// TwinCAT 3 PLC project main_program
// ProgramVersion: 3.1.4024.0
// libraries:
//   Tc2_MC2, * (Beckhoff Automation GmbH)
//   Tc2_Utilities, * (Beckhoff Automation GmbH)
//   Tc2_Standard, * (Beckhoff Automation GmbH)
//   Tc2_System, * (Beckhoff Automation GmbH)
//   Tc3_Module, * (Beckhoff Automation GmbH)
// project tree:
//   DUTs/ E_BiaxialState.TcDUT, E_PlcSystemStatus.TcDUT, E_SafetyState.TcDUT, E_SyncPoint.TcDUT, ST_settings.TcDUT (not stored), ST_MoveCommand.TcDUT, ST_SystemStatus.TcDUT
//   GVLs/ GVL_Axis.TcGVL (not stored), GVL_Persistent.TcGVL
//   / PlcTask.TcTTO (not stored)
//   POUs/ fb_MovementController.TcPOU, fb_AxisStatusPublisher.TcPOU, fb_BiaxialCoordinator.TcPOU, fb_safety.TcPOU, fb_StatusBuffer.TcPOU, MAIN.TcPOU
// real-time tasks:
//   TASK PlcTask: cycle T#10ms, priority 20, ADS port 350
// motion (NC):
//   TASK NC-Task 1 SAF: cycle T#2ms, priority 4, ADS port 501
//   TASK NC-Task 1 SVB: cycle T#10ms, priority 8, ADS port 511
//   AXIS xAxis (id 1)
//     Dynamic: Acceleration=150, Deceleration=150, Jerk=225
//     Velo: RefSearch=2, RefSync=5, SlowManual=5, FastManual=10, Maximum=100
//     OtherSettings: AllowMotionCmdToSlave=true
//     encoder EncType=19
//       EncPara: ScaleFactorNumerator=2, ScaleFactorDenominator=1048576, MaxCount=#xffffffff
//         SoftEndMaxControl: Range=10000
//         Inc: RefSearchInverse=true, RefPosition=-5
//     drive DrvType=16
//       DrvPara: MaxCount=#xffffffff, DriveControlDWord=#x00020100
//         Analog: TorqueSetpointScale=10, ScaleFactorActTorque=0.1
//         TimeComp: TaskDelayCycles=1
//     controller CtrType=1
//       CtrPara: PriorControlFactor=1
//         Observer: BandWidth=20
//   AXIS yAxis (id 2)
//     Dynamic: Acceleration=150, Deceleration=150, Jerk=225
//     Velo: RefSearch=2, RefSync=5, SlowManual=5, FastManual=10, Maximum=100
//     OtherSettings: AllowMotionCmdToSlave=true
//     encoder EncType=19
//       EncPara: ScaleFactorNumerator=2, ScaleFactorDenominator=1048576, MaxCount=#xffffffff
//         SoftEndMinControl: Enable=true
//         SoftEndMaxControl: Range=10000
//         Inc: RefSearchInverse=true, RefPosition=-5, RefMode=1
//     drive DrvType=16
//       DrvPara: MaxCount=#xffffffff, DriveControlDWord=#x00020100
//         Analog: TorqueSetpointScale=10, ScaleFactorActTorque=0.1
//         TimeComp: TaskDelayCycles=1
//     controller CtrType=1
//       CtrPara: PriorControlFactor=1
//         Observer: BandWidth=20
// I/O:
//   DEVICE Device 1 (EtherCAT), AmsNetId 5.85.113.174.2.1
//     Term 1 (EK1200) [EK1200-5000 EtherCAT Power supply (2A E-Bus)]
//       Term 2 (EL7062) [EL7062-0000 2Ch. Stepper motor output stage (48V, 3A)]
//       Term 3 (EL9510) [EL9510 Power supply terminal 10V]
//       Term 4 (EL3356-0020) [EL3356-0020 1Ch. Ana. Input Resistor Bridge Terminal, 24bit, High Precision, with calibration certificate]
//       Term 5 (EL3356-0020) [EL3356-0020 1Ch. Ana. Input Resistor Bridge Terminal, 24bit, High Precision, with calibration certificate]
//       Term 6 (EL9011) [EL9011 End Terminal]
// variable links:
//   NC-Task 1 SAF/Axes/xAxis <-> Device 1 (EtherCAT)/Term 1 (EK1200)/Term 2 (EL7062)
//     Drive/Inputs/In/nDataIn1 <-> DRV Following error actual value Channel 2/Following error actual value
//     Drive/Inputs/In/nDcOutputTime <-> InfoData/DcOutputShift
//     Drive/Inputs/In/nState1 <-> DRV Statusword Channel 2/Statusword
//     Drive/Inputs/In/nState2 <-> DRV Statusword Channel 2/Statusword @bit 8
//     Drive/Inputs/In/nState4 @bit 1 <-> WcState/InputToggle
//     Drive/Inputs/In/nState4 <-> WcState/WcState
//     Drive/Outputs/Out/nCtrl1 <-> DRV Controlword Channel 2/Controlword
//     Drive/Outputs/Out/nCtrl2 <-> DRV Controlword Channel 2/Controlword @bit 8
//     Drive/Outputs/Out/nDataOut1 <-> DRV Target position Channel 2/Target position
//     Enc/Inputs/In/nDataIn1 <-> FB Position Channel 2/Position
//     Enc/Inputs/In/nDcInputTime <-> InfoData/DcInputShift
//     Enc/Inputs/In/nState4 @bit 1 <-> WcState/InputToggle
//     Enc/Inputs/In/nState4 <-> WcState/WcState
//   NC-Task 1 SAF/Axes/yAxis <-> Device 1 (EtherCAT)/Term 1 (EK1200)/Term 2 (EL7062)
//     Drive/Inputs/In/nDataIn1 <-> DRV Following error actual value Channel 1/Following error actual value
//     Drive/Inputs/In/nDcOutputTime <-> InfoData/DcOutputShift
//     Drive/Inputs/In/nState1 <-> DRV Statusword Channel 1/Statusword
//     Drive/Inputs/In/nState2 <-> DRV Statusword Channel 1/Statusword @bit 8
//     Drive/Inputs/In/nState4 @bit 1 <-> WcState/InputToggle
//     Drive/Inputs/In/nState4 <-> WcState/WcState
//     Drive/Outputs/Out/nCtrl1 <-> DRV Controlword Channel 1/Controlword
//     Drive/Outputs/Out/nCtrl2 <-> DRV Controlword Channel 1/Controlword @bit 8
//     Drive/Outputs/Out/nDataOut1 <-> DRV Target position Channel 1/Target position
//     Enc/Inputs/In/nDataIn1 <-> FB Position Channel 1/Position
//     Enc/Inputs/In/nDcInputTime <-> InfoData/DcInputShift
//     Enc/Inputs/In/nState4 @bit 1 <-> WcState/InputToggle
//     Enc/Inputs/In/nState4 <-> WcState/WcState
//   main program/main program Instance <-> Device 1 (EtherCAT)/Term 1 (EK1200)/Term 2 (EL7062)
//     PlcTask Inputs/MAIN.nEndStopHx <-> DI Inputs Channel 2/Input 1
//     PlcTask Inputs/MAIN.nEndStopHy <-> DI Inputs Channel 1/Input 2
//     PlcTask Inputs/MAIN.nEndStopLx <-> DI Inputs Channel 1/Input 1
//     PlcTask Inputs/MAIN.nEndStopLy <-> DI Inputs Channel 2/Input 2
//   main program/main program Instance <-> Device 1 (EtherCAT)/Term 1 (EK1200)/Term 4 (EL3356-0020)
//     PlcTask Inputs/MAIN.nRawTenzoX <-> RMB Value (INT32)/Value
//   main program/main program Instance <-> Device 1 (EtherCAT)/Term 1 (EK1200)/Term 5 (EL3356-0020)
//     PlcTask Inputs/MAIN.nRawTenzoY <-> RMB Value (INT32)/Value
//   main program/main program Instance <-> NC-Task 1 SAF/Axes/xAxis
//     PlcTask Inputs/GVL_Axis.xAxis.NcToPlc <-> Outputs/ToPlc
//     PlcTask Outputs/GVL_Axis.xAxis.PlcToNc <-> Inputs/FromPlc
//   main program/main program Instance <-> NC-Task 1 SAF/Axes/yAxis
//     PlcTask Inputs/GVL_Axis.yAxis.NcToPlc <-> Outputs/ToPlc
//     PlcTask Outputs/GVL_Axis.yAxis.PlcToNc <-> Inputs/FromPlc

// ---- DUTs/E_BiaxialState.TcDUT
{attribute 'qualified_only'}
TYPE E_BiaxialState :
(
	Idle,
	Running,
	Aborting,
	Completing
);
END_TYPE

// ---- DUTs/E_PlcSystemStatus.TcDUT
{attribute 'qualified_only'}
TYPE E_PlcSystemStatus :
(
	Idle := 0,
	Error := 1,
	Homing := 2,
	Stopping := 3,
	Taring := 4,
	BasicMove := 5,
	ForceMode := 6,
	Pretension := 10,
	PreTestCyclic := 11,
	SingleTest := 20,
	CyclicTest := 21,
	PostTest := 30
);
END_TYPE

// ---- DUTs/E_SafetyState.TcDUT
TYPE E_SafetyState :
(
	Idle,
	RestoreReference,
	VerifyReference,
	Homing,
	MoveToZero,
	Complete,
	ProtectiveStop,
	ErrorStop
);
END_TYPE

// ---- DUTs/E_SyncPoint.TcDUT
{attribute 'qualified_only'}
TYPE E_SyncPoint :
(
	None := 0,
	PreTestDone := 1,
	LoadDone := 2,
	UnloadDone := 3,
	MainDone := 4,
	PostTestDone := 5,
	PretensionDone := 6
);
END_TYPE

// ---- DUTs/ST_MoveCommand.TcDUT
TYPE ST_MoveCommand :
	STRUCT
		// Mode 1: maintained jog
		fMoveVelocity : LREAL; // Signed jog velocity while bExecute is TRUE
		nJogLeaseCounter : UDINT; // Must change periodically while a jog is held

		// Mode 2: one PI-regulated force hold
		fTargetForce   : LREAL;
		fForceDuration : LREAL;
	
		// Command and service controls
		nMode       : INT;  // 1=jog, 2=force/time, 3=test sequence
		bExecute    : BOOL; // Start movement; maintained press signal for jog
		bHalt       : BOOL; // Panic stop
		bPower      : BOOL; // Maintained motor-enable request
		bReset      : BOOL; // Reset errors
		bHome       : BOOL; // Start homing sequence
		bStartTar   : BOOL; // Start tare sequence
		bSavePosition : BOOL; // Capture the current axis position while idle
		bRestorePosition : BOOL; // Return to the saved coordinate while idle
		fRestoreVelocity : LREAL; // Saved-position return speed [mm/s]

		// Optional force pre-conditioning sequence
		bIncludePreTest : BOOL;
		bPreTestOnly    : BOOL;  // Run pre-test and post-test without a main test
		nPreCycleCount  : INT;   // Number of force load/unload cycles, 0..50
		bPreloadEnabled : BOOL;  // Apply one force preload before the first cycle
		fPreloadValue   : LREAL; // Signed preload force [N]
		fPreCycleLoadValue : LREAL; // Signed repeated preconditioning load target [N]
		fPreUnloadValue : LREAL; // Signed force unload target [N]
		bPreUnloadToStart : BOOL; // Return to sequence-start position instead of force unload
		fPreTestRate     : LREAL; // Positive motor speed magnitude [mm/s]
		fPreTestForceTolerance : LREAL := 0.1; // [N], or negative for target-relative percent
		fPreloadHoldTime : LREAL := 0.0; // Hold time for the initial preload endpoint [s]
		fPreCycleHoldTime : LREAL := 0.0; // Hold time for cyclic pre-conditioning endpoints [s]

		// Main test settings
		fTestRate      : LREAL; // Positive motor speed magnitude [mm/s]
		fSingleForceTolerance : LREAL := 0.1; // [N], or negative for target-relative percent
		fSingleForceHoldTime : LREAL := 0.0; // Hold time for the single-test primary endpoint [s]
		fCyclicForceTolerance : LREAL := 0.1; // [N], or negative for target-relative percent
		fCyclicForceHoldTime : LREAL := 0.0; // Hold time for cyclic load/unload endpoints [s]

		// Test selection: >0=cyclic count, 0=single test
		nCycleCount : INT;
		nLoadMode   : INT;   // 1=displacement, 2=force
		fLoadValues : ARRAY[1..50] OF LREAL; // per-cycle level [mm] or signed force [N]
		nUnloadMode : INT;   // 1=displacement, 2=force
		fUnloadValues : ARRAY[1..50] OF LREAL; // per-cycle level [mm] or signed force [N]

		// Single test (nMode=3, nCycleCount=0); criterion 2 is optional OR
		nStop1Mode         : INT;   // 0=off, 1=displacement, 2=force
		fStop1Value        : LREAL;
		nStop2Mode         : INT;   // 0=off, 1=displacement, 2=force, 3=rupture
		fStop2Value        : LREAL;

		// 0=stay, 1=saved position, 2=sequence start,
		// 3=pre-test final position, 4=unload to zero force
		nPostTestMode : INT;
	END_STRUCT
END_TYPE

// ---- DUTs/ST_SystemStatus.TcDUT
TYPE ST_SystemStatus :
	STRUCT
		fPosBuffer   : ARRAY[1..50] OF LREAL; // Circular display-position samples
		fTenzoBuffer : ARRAY[1..50] OF LREAL; // Circular force samples
		nBufferHead  : INT := 50;             // Index of latest completely written sample
		nSampleCounter    : UDINT := 0;       // Wrapping sample counter for drop detection
		nOperationCounter : UDINT := 0;       // Incremented after each completed motion command
		nInterfaceVersion : UDINT := 7;       // MATLAB/PLC ADS contract version
		fTenzoTarOffset   : LREAL := 0.0;     // Calculated tar offset
		fActPosition : LREAL := 0.0;          // Display position (50 mm - NC position)
		
		bWorking     : BOOL;                   // PLC occupied; do not send a new test
		bTarWorking  : BOOL;                   // PLC is calculating tare
		bError       : BOOL;                   // Latched application or motion error
		nErrorCode   : UDINT := 0;             // Application error code (0 = no error)
		nAxisErrorID : UDINT := 0;             // Native TwinCAT/NC error ID
		bPowered     : BOOL;                   // Axis power is enabled
		bHoming      : BOOL;                   // Homing command is active
		bHomed       : BOOL;                   // NC axis reports a valid home reference
		bStopped     : BOOL;                   // Axis is at standstill
		bSavedPositionValid : BOOL;            // A return-to-saved reference is available
		nSystemStatus : INT := 0;              // High-level numeric system status
	END_STRUCT
END_TYPE

// ---- GVLs/GVL_Persistent.TcGVL
{attribute 'qualified_only'}
VAR_GLOBAL PERSISTENT
	// Last valid incremental-axis coordinates
	fLastPositionX      : LREAL;
	fLastPositionY      : LREAL;
	bLastPositionValidX : BOOL;
	bLastPositionValidY : BOOL;
END_VAR

// ---- POUs/fb_MovementController.TcPOU
FUNCTION_BLOCK fb_MovementController
VAR_INPUT
	fForce        : LREAL; // Actual force
	fActPosition  : LREAL; // Absolute NC position
	bPowerState   : BOOL;  // Actual power on state
	bHaltDone     : BOOL;  // Motor stopped
	bAxisStopped  : BOOL;  // Fresh safety/NC standstill state
	bSafetyError  : BOOL;
	bProtectiveStop : BOOL;
	bExternalBusy : BOOL;
	bReferenceValid : BOOL; // Current home/reference belongs to this coordinate system
	bInvalidateSavedPosition : BOOL; // Home request invalidates saved absolute coordinates
	bSyncEnabled  : BOOL;  // TRUE only for a PLC-owned biaxial test
	bSyncRelease  : BOOL;  // Shared barrier release from MAIN
	bSyncAbort    : BOOL;  // Stop this axis when the synchronized peer aborts
	bSyncSingleComplete : BOOL; // Peer reached its biaxial Single endpoint
	stSettings    : ST_Settings;
END_VAR

VAR_OUTPUT
	fTestStartPos : LREAL := 0.0; // position where test started
	stateHalt   : BOOL; // Request a controlled stop
	bBusy       : BOOL; // System is processing a test or stopping
	bError      : BOOL; // Latched application/motion error
	nErrorCode  : UDINT;
	nAxisErrorID: UDINT;
	nOperationCounter : UDINT;
	bSavedPositionValid : BOOL;
	nSystemStatus : INT; // High-level numeric system status exposed through ADS
	nSyncPoint : BYTE; // E_SyncPoint: 0 none through 6 pretension
	nSyncCycle : INT;  // Cycle associated with the current sync point
	bPeerAbortRequest : BOOL; // Abort synchronized peer while local relief continues
END_VAR

VAR
	// Movement FBs
	fbMC_MoveRelative1 : MC_MoveRelative;
	fbMC_MoveVelocity  : MC_MoveVelocity;
	
	// Shared help vars
	nSeqState    : INT; // Current sequence state
	
	// mode 1
	fTargetDist1 : LREAL;
	fTargetVel1  : LREAL;
	
	// mode 2/3 vel movement
	bExecuteVelMove : BOOL;
    fCmdVelocity    : LREAL;
    mcDirection     : MC_Direction;
	
	// mode 2/3 help vars
	fTargetForce          : LREAL; // Wanted F
    fForceError           : LREAL; // Regulation error
    fForceErrorIntegral   : LREAL; // Integ of error
	fMode2HoldElapsed     : LREAL; // Accumulated time inside force tolerance
	fLastSentVelocity   : LREAL;    // Tracks last updated velocity to prevent NC spamming
	fPendingVelocity   : LREAL;
	mcPendingDirection : MC_Direction;
	nVelocityState     : INT;
	nVelocityUpdateCounter : INT;
	fForceRegMaxVelocity : LREAL; // Mode-3 P regulator speed limit
	fForceRegMinVelocity : LREAL; // Mode-3 low-speed hold deadband
	bResetRequested : BOOL;
	bOperationCompleted : BOOL;

	// Saved/reference positions
	fSavedPosition      : LREAL;
	fPreTestFinalPos    : LREAL;
	rtSavePosition      : R_TRIG;
	rtRestorePosition   : R_TRIG;
	rtSyncAbort         : R_TRIG;
	fbJogLease          : TON;
	nLastJogLeaseCounter : UDINT;
	bJogLeaseRenewed    : BOOL;

	// Generic endpoint engine for test-sequence mode 3
	nCurrentCycle           : INT;
	nCurrentPreCycle        : INT;
	nAfterEndpointState     : INT;
	fEndpointTargetPosition : LREAL;
	fEndpointTargetForce    : LREAL;
	fEndpointRate           : LREAL;
	fEndpointTolerance      : LREAL;
	fEndpointHoldTime       : LREAL;
	fEndpointStartError     : LREAL;
	fEndpointCurrentError   : LREAL;
	fForceHoldElapsed       : LREAL;
	fPositionHoldElapsed    : LREAL;
	nLoadDirection          : INT;
	nLastMotionDirection    : INT;
	nReliefSourceDirection  : INT;
	nEndpointSyncPoint      : BYTE;
	nEndpointSyncCycle      : INT;
	bForceEndpointReady     : BOOL;
	bZeroForceUnload        : BOOL; // Post-test unload must not reverse across zero

	// Optional OR criterion for the single test
	bSinglePrimaryActive  : BOOL;
	bSingleStopReached    : BOOL;
	fStop2TargetPosition  : LREAL;
	fStop2StartError      : LREAL;
	fStop2CurrentError    : LREAL;
	fSingleStartForce     : LREAL;
	fSinglePeakForce      : LREAL;
	bSingleRuptureArmed   : BOOL;
	
END_VAR

VAR CONSTANT
	// Task and controller constants
	CYCLE_TIME : LREAL := 0.01; // dt of plc
	VELOCITY_UPDATE_DELTA : LREAL := 0.1;
	VELOCITY_UPDATE_CYCLES : INT := 10;
	FORCE_REG_MIN_SPEED_FRACTION : LREAL := 0.01;
	POSITION_EPSILON : LREAL := 0.000001;
	FORCE_POLARITY : INT := -1;
	STATUS_IDLE : INT := 0;
	STATUS_STOPPING : INT := 3;
	STATUS_BASIC_MOVE : INT := 5;
	STATUS_FORCE_MODE : INT := 6;
	STATUS_PRETENSION : INT := 10;
	STATUS_PRETEST_CYCLIC : INT := 11;
	STATUS_SINGLE_TEST : INT := 20;
	STATUS_CYCLIC_TEST : INT := 21;
	STATUS_POSTTEST : INT := 30;
	SYNC_NONE : BYTE := 0;
	SYNC_PRETEST_DONE : BYTE := 1;
	SYNC_LOAD_DONE : BYTE := 2;
	SYNC_UNLOAD_DONE : BYTE := 3;
	SYNC_MAIN_DONE : BYTE := 4;
	SYNC_POSTTEST_DONE : BYTE := 5;
	SYNC_PRETENSION_DONE : BYTE := 6;
	STATE_IDLE : INT := 0;
	STATE_MODE_START : INT := 1;
	STATE_MODE_RUN : INT := 2;
	STATE_PRELOAD : INT := 10;
	STATE_CAPTURE_TEST_START : INT := 11;
	STATE_PRE_CYCLE_LOAD : INT := 12;
	STATE_PRE_CYCLE_UNLOAD : INT := 13;
	STATE_PRE_CYCLE_NEXT : INT := 14;
	STATE_CAPTURE_PRETEST_FINAL : INT := 18;
	STATE_PRETEST_BARRIER : INT := 19;
	STATE_SELECT_MAIN_TEST : INT := 20;
	STATE_SECONDARY_BARRIER : INT := 49;
	STATE_POSTTEST_SELECT : INT := 50;
	STATE_POSTTEST_WAIT_STOP : INT := 51;
	STATE_POSTTEST_BARRIER : INT := 54;
	STATE_OPERATION_COMPLETE : INT := 55;
	STATE_RESTORE_COMPLETE : INT := 56;
	STATE_CYCLIC_LOAD : INT := 100;
	STATE_CYCLIC_UNLOAD : INT := 110;
	STATE_CYCLIC_NEXT : INT := 120;
	STATE_CYCLIC_COMPLETE : INT := 121;
	STATE_SINGLE_START : INT := 200;
	STATE_SINGLE_WAIT_STOP : INT := 220;
	STATE_POSITION_PREPARE : INT := 300;
	STATE_POSITION_EXECUTE : INT := 301;
	STATE_POSITION_WAIT : INT := 302;
	STATE_POSITION_HOLD : INT := 303;
	STATE_POSITION_BARRIER : INT := 304;
	STATE_FORCE_PREPARE : INT := 310;
	STATE_FORCE_EXECUTE : INT := 311;
	STATE_FORCE_WAIT_TOLERANCE : INT := 312;
	STATE_FORCE_WAIT_STOP : INT := 313;
	STATE_FORCE_HOLD : INT := 314;
	STATE_FORCE_EXIT_WAIT_STOP : INT := 315;
	STATE_FORCE_READY_WAIT_STOP : INT := 316;
	STATE_ABORT_STOPPING : INT := 900;
	STATE_RELIEF_WAIT_STOP : INT := 910;
	STATE_RELIEF_START : INT := 911;
	STATE_RELIEF_WAIT_MOVE : INT := 912;
	STATE_ERROR_STOPPING : INT := 998;
	STATE_ERROR_LATCHED : INT := 999;
	ERROR_UNSUPPORTED_MODE : UDINT := 2001;
	ERROR_SAVED_POSITION_UNAVAILABLE : UDINT := 2002;
	ERROR_UNSUPPORTED_ENDPOINT : UDINT := 2003;
	ERROR_UNSUPPORTED_POST_ACTION : UDINT := 2005;
	ERROR_POWER_UNAVAILABLE : UDINT := 2006;
	ERROR_INVALID_CONFIGURATION : UDINT := 2007;
	ERROR_COMMAND_CONFLICT : UDINT := 2008;
	ERROR_INVALID_RUNTIME_VALUE : UDINT := 2009;
	ERROR_JOG_LEASE_EXPIRED : UDINT := 2011;
	ERROR_VELOCITY_LIMIT : UDINT := 2012;
	ERROR_RELIEF_COMPLETED : UDINT := 2101;
	ERROR_RELIEF_DIRECTION_UNKNOWN : UDINT := 2102;
	ERROR_RELATIVE_MOVE : UDINT := 2201;
	ERROR_VELOCITY_MOVE : UDINT := 2203;
END_VAR

VAR_IN_OUT
	Axis          : AXIS_REF;
	stMoveCommand : ST_MoveCommand;
END_VAR


// =========================================================
//                    Saved position
// =========================================================

rtSavePosition(CLK := stMoveCommand.bSavePosition);
rtRestorePosition(CLK := stMoveCommand.bRestorePosition);
rtSyncAbort(CLK := bSyncEnabled AND bSyncAbort);

// Saved positions are absolute NC coordinates. A new home/reference changes
// their meaning, so discard them as soon as homing starts or reference is lost.
IF bInvalidateSavedPosition OR NOT bReferenceValid THEN
	bSavedPositionValid := FALSE;
END_IF

IF rtSavePosition.Q AND nSeqState = STATE_IDLE AND NOT bExternalBusy AND
	bReferenceValid AND bAxisStopped THEN
	fSavedPosition := fActPosition;
	bSavedPositionValid := TRUE;
END_IF

// A maintained jog must be renewed by the ADS owner. The monotonically
// increasing counter makes a stale TRUE bExecute harmless after owner loss.
bJogLeaseRenewed := nSeqState = STATE_MODE_RUN AND
	stMoveCommand.nMode = 1 AND
	stMoveCommand.nJogLeaseCounter <> nLastJogLeaseCounter;
IF bJogLeaseRenewed THEN
	nLastJogLeaseCounter := stMoveCommand.nJogLeaseCounter;
END_IF
fbJogLease(
	IN := nSeqState = STATE_MODE_RUN AND stMoveCommand.nMode = 1 AND
		NOT bJogLeaseRenewed,
	PT := T#750MS);
IF fbJogLease.Q AND NOT bError AND NOT bSafetyError THEN
	stMoveCommand.bExecute := FALSE;
	SetError(
		nCode := ERROR_JOG_LEASE_EXPIRED,
		nNativeErrorID := 0,
		bRequestHalt := TRUE);
END_IF

// =========================================================
//                      Error handling
// =========================================================

IF stMoveCommand.bReset THEN
	bResetRequested := TRUE;
END_IF

IF bResetRequested AND bError AND NOT bSafetyError THEN
	bError := FALSE;
	nErrorCode := 0;
	nAxisErrorID := 0;
	nSeqState := STATE_IDLE;
	stateHalt := FALSE;
	bResetRequested := FALSE;
ELSIF bResetRequested AND NOT bError AND NOT bSafetyError THEN
	IF nSeqState = STATE_ERROR_LATCHED THEN
		nSeqState := STATE_IDLE;
	END_IF
	bResetRequested := FALSE;
END_IF

// Operator and safety stops abort the sequence without running post-test.
IF stMoveCommand.bHalt OR (bProtectiveStop AND NOT stateHalt) OR
	rtSyncAbort.Q THEN
	IF stMoveCommand.bHalt THEN
		stMoveCommand.bHalt := FALSE;
	END_IF
	stMoveCommand.bExecute := FALSE;
	ClearActiveCommand();
	stateHalt := TRUE;
	nSeqState := STATE_ABORT_STOPPING;
END_IF

// A safety-owned error cancels local motion without issuing another halt.
IF bSafetyError THEN
	stMoveCommand.bExecute := FALSE;
	ClearActiveCommand();
	stateHalt := FALSE;
	nSeqState := STATE_ERROR_LATCHED;
END_IF

// Latch motion-function-block and sensor errors.
IF NOT bError AND NOT bSafetyError THEN
	IF fbMC_MoveRelative1.Error THEN
		bError := TRUE;
		nErrorCode := ERROR_RELATIVE_MOVE;
		nAxisErrorID := fbMC_MoveRelative1.ErrorID;
	ELSIF fbMC_MoveVelocity.Error THEN
		bError := TRUE;
		nErrorCode := ERROR_VELOCITY_MOVE;
		nAxisErrorID := fbMC_MoveVelocity.ErrorID;
	ELSIF nSeqState > STATE_IDLE AND
		nSeqState < STATE_ABORT_STOPPING AND
		NOT ((fForce = fForce) AND ABS(fForce) < 1.0E300) THEN
		bError := TRUE;
		nErrorCode := ERROR_INVALID_RUNTIME_VALUE;
	END_IF
END_IF

// Runtime overforce response: halt, make one fixed relative release move, then abort.
IF NOT bError AND NOT bSafetyError AND
	nSeqState > STATE_IDLE AND nSeqState < STATE_ABORT_STOPPING AND
	ABS(fForce) >= stSettings.fMaxForce THEN
	IF Axis.Status.PositiveDirection THEN
		nReliefSourceDirection := 1;
	ELSIF Axis.Status.NegativeDirection THEN
		nReliefSourceDirection := -1;
	ELSIF stMoveCommand.nMode = 3 AND nLoadDirection <> 0 THEN
		nReliefSourceDirection := nLoadDirection;
	ELSE
		nReliefSourceDirection := nLastMotionDirection;
	END_IF
	fbMC_MoveRelative1.Execute := FALSE;
	bExecuteVelMove := FALSE;
	bSinglePrimaryActive := FALSE;
	bForceEndpointReady := FALSE;
	nSyncPoint := SYNC_NONE;
	nSyncCycle := 0;
	stateHalt := TRUE;
	nSeqState := STATE_RELIEF_WAIT_STOP;
END_IF

IF bError AND nSeqState <> STATE_ERROR_STOPPING AND
	nSeqState <> STATE_ERROR_LATCHED THEN
	stMoveCommand.bExecute := FALSE;
	ClearActiveCommand();
	stateHalt := TRUE;
	nSeqState := STATE_ERROR_STOPPING;
END_IF

IF bError THEN
	stMoveCommand.bExecute := FALSE;
END_IF

IF stMoveCommand.bExecute AND bExternalBusy THEN
	stMoveCommand.bExecute := FALSE;
	bError := TRUE;
	nErrorCode := ERROR_COMMAND_CONFLICT;
END_IF

IF stMoveCommand.bExecute AND NOT bPowerState THEN
	stMoveCommand.bExecute := FALSE;
	bError := TRUE;
	nErrorCode := ERROR_POWER_UNAVAILABLE;
END_IF

// Finish operator/error stops.
IF (nSeqState = STATE_ABORT_STOPPING OR
	nSeqState = STATE_ERROR_STOPPING) AND bHaltDone THEN
	stateHalt := FALSE;
	IF nSeqState = STATE_ERROR_STOPPING THEN
		nSeqState := STATE_ERROR_LATCHED;
	ELSE
		nSeqState := STATE_IDLE;
	END_IF
END_IF

// Overforce release sequence. FB1 is reused with aborting buffer mode.
CASE nSeqState OF
	STATE_RELIEF_WAIT_STOP:
		IF bHaltDone THEN
			stateHalt := FALSE;
			IF nReliefSourceDirection = 0 THEN
				bError := TRUE;
				nErrorCode := ERROR_RELIEF_DIRECTION_UNKNOWN;
				nSeqState := STATE_ERROR_LATCHED;
			ELSE
				fTargetDist1 := -INT_TO_LREAL(nReliefSourceDirection) *
					ABS(stSettings.fForceReliefDistance);
				fTargetVel1 := ABS(stSettings.fForceReliefVelocity);
				fbMC_MoveRelative1.Execute := FALSE;
				nSeqState := STATE_RELIEF_START;
			END_IF
		END_IF

	STATE_RELIEF_START:
		fbMC_MoveRelative1.Execute := TRUE;
		nSeqState := STATE_RELIEF_WAIT_MOVE;

	STATE_RELIEF_WAIT_MOVE:
		IF fbMC_MoveRelative1.Done THEN
			fbMC_MoveRelative1.Execute := FALSE;
			bError := TRUE;
			nErrorCode := ERROR_RELIEF_COMPLETED;
			nAxisErrorID := 0;
			nSeqState := STATE_ERROR_LATCHED;
		END_IF
END_CASE

// Saved-position restore is a service operation and is independent of nMode.
IF rtRestorePosition.Q AND nSeqState = STATE_IDLE AND
	NOT bError AND NOT bSafetyError THEN
	IF bExternalBusy THEN
		stMoveCommand.bExecute := FALSE;
		SetError(
			nCode := ERROR_COMMAND_CONFLICT,
			nNativeErrorID := 0,
			bRequestHalt := TRUE);
	ELSIF NOT bPowerState THEN
		stMoveCommand.bExecute := FALSE;
		SetError(
			nCode := ERROR_POWER_UNAVAILABLE,
			nNativeErrorID := 0,
			bRequestHalt := TRUE);
	ELSIF NOT bReferenceValid OR NOT bSavedPositionValid THEN
		stMoveCommand.bExecute := FALSE;
		SetError(
			nCode := ERROR_SAVED_POSITION_UNAVAILABLE,
			nNativeErrorID := 0,
			bRequestHalt := TRUE);
	ELSIF NOT ((stMoveCommand.fRestoreVelocity =
		stMoveCommand.fRestoreVelocity) AND
		ABS(stMoveCommand.fRestoreVelocity) > 0.0 AND
		ABS(stMoveCommand.fRestoreVelocity) < 1.0E300) THEN
		stMoveCommand.bExecute := FALSE;
		SetError(
			nCode := ERROR_INVALID_RUNTIME_VALUE,
			nNativeErrorID := 0,
			bRequestHalt := TRUE);
	ELSIF ABS(stMoveCommand.fRestoreVelocity) > ABS(stSettings.fMaxVelocity) THEN
		stMoveCommand.bExecute := FALSE;
		SetError(
			nCode := ERROR_VELOCITY_LIMIT,
			nNativeErrorID := 0,
			bRequestHalt := TRUE);
	ELSE
		fTestStartPos := fActPosition;
		nSystemStatus := STATUS_BASIC_MOVE;
		nLoadDirection := 0;
		nLastMotionDirection := 0;
		nReliefSourceDirection := 0;
		PreparePositionEndpoint(
			fTargetPosition := fSavedPosition,
			fRate := stMoveCommand.fRestoreVelocity,
			fHoldTime := 0.0,
			nTargetSyncPoint := SYNC_NONE,
			nTargetSyncCycle := 0,
			nNextState := STATE_RESTORE_COMPLETE);
	END_IF
END_IF

// =========================================================
//                      Mode switcher
// =========================================================

// In a biaxial Single test, either axis endpoint completes both axes.
IF bSinglePrimaryActive AND bSyncSingleComplete THEN
	fbMC_MoveRelative1.Execute := FALSE;
	bExecuteVelMove := FALSE;
	bSinglePrimaryActive := FALSE;
	stateHalt := TRUE;
	nSeqState := STATE_SINGLE_WAIT_STOP;
END_IF

IF NOT bError AND NOT bSafetyError AND
	nSeqState < STATE_ABORT_STOPPING THEN
	IF nSeqState >= STATE_POSITION_PREPARE AND
		nSeqState <= STATE_POSITION_BARRIER THEN
		positionEndpoint();
	ELSIF nSeqState >= STATE_FORCE_PREPARE AND
		nSeqState <= STATE_FORCE_READY_WAIT_STOP THEN
		forceEndpoint();
	ELSIF nSeqState = STATE_RESTORE_COMPLETE THEN
		testSequence();
	ELSE
		CASE stMoveCommand.nMode OF
			1: mode1();
			2: mode2();
			3: testSequence();
		ELSE
			IF stMoveCommand.bExecute THEN
				stMoveCommand.bExecute := FALSE;
				bError := TRUE;
				nErrorCode := ERROR_UNSUPPORTED_MODE;
			END_IF
		END_CASE
	END_IF
END_IF

// =========================================================
//                      Motion calls
// =========================================================

fbMC_MoveRelative1(
	Axis := Axis,
	Distance := fTargetDist1,
	Velocity := MIN(ABS(fTargetVel1), ABS(stSettings.fMaxVelocity)),
	BufferMode := MC_Aborting);

fbMC_MoveVelocity(
	Axis := Axis,
	Execute := bExecuteVelMove,
	Velocity := MIN(ABS(fCmdVelocity), ABS(stSettings.fMaxVelocity)),
	Direction := mcDirection,
	BufferMode := MC_Aborting);

IF Axis.Status.PositiveDirection THEN
	nLastMotionDirection := 1;
ELSIF Axis.Status.NegativeDirection THEN
	nLastMotionDirection := -1;
END_IF

// =========================================================
//                         Outputs
// =========================================================

IF nSeqState = STATE_IDLE THEN
	nSystemStatus := STATUS_IDLE;
ELSIF nSeqState >= STATE_ABORT_STOPPING THEN
	nSystemStatus := STATUS_STOPPING;
END_IF

// Expose a newly entered relief state in this scan
bPeerAbortRequest := nSeqState >= STATE_RELIEF_WAIT_STOP AND
	nSeqState <= STATE_RELIEF_WAIT_MOVE;

bBusy := nSeqState > STATE_IDLE AND
	nSeqState <> STATE_ERROR_LATCHED;

IF bOperationCompleted THEN
	nOperationCounter := nOperationCounter + 1;
	bOperationCompleted := FALSE;
END_IF

METHOD ClearActiveCommand

fbMC_MoveRelative1.Execute := FALSE;
bExecuteVelMove := FALSE;
bSinglePrimaryActive := FALSE;
bForceEndpointReady := FALSE;
bZeroForceUnload := FALSE;
fPositionHoldElapsed := 0.0;
nSyncPoint := SYNC_NONE;
nSyncCycle := 0;
END_METHOD

ACTION forceEndpoint:

CASE nSeqState OF
	STATE_FORCE_PREPARE:
		bExecuteVelMove := FALSE;
		fForceHoldElapsed := 0.0;
		bForceEndpointReady := FALSE;
		nSyncPoint := SYNC_NONE;
		nSyncCycle := 0;
		fEndpointStartError := fEndpointTargetForce - fForce;
		nVelocityState := 0;
		nVelocityUpdateCounter := VELOCITY_UPDATE_CYCLES;
		fLastSentVelocity := 0.0;
		fForceRegMaxVelocity := MIN(
			ABS(fEndpointRate),
			ABS(stSettings.fMaxVelocity));
		// Keep the anti-chatter floor small enough that force endpoints settle
		// near the requested goal instead of at the edge of a 10% speed band.
		fForceRegMinVelocity := fForceRegMaxVelocity *
			FORCE_REG_MIN_SPEED_FRACTION;
		fCmdVelocity := ABS(fEndpointRate);
		IF fEndpointStartError * INT_TO_LREAL(FORCE_POLARITY) >= 0.0 THEN
			mcDirection := MC_Positive_Direction;
			nLoadDirection := 1;
			nLastMotionDirection := 1;
		ELSE
			mcDirection := MC_Negative_Direction;
			nLoadDirection := -1;
			nLastMotionDirection := -1;
		END_IF
		IF ABS(fEndpointStartError) <= fEndpointTolerance THEN
			stateHalt := TRUE;
			nVelocityState := 3;
			nSeqState := STATE_FORCE_WAIT_STOP;
		ELSE
			nSeqState := STATE_FORCE_EXECUTE;
		END_IF

	STATE_FORCE_EXECUTE: // Trigger constant-speed force approach.
		bExecuteVelMove := TRUE;
		nVelocityState := 1;
		nSeqState := STATE_FORCE_WAIT_TOLERANCE;

	STATE_FORCE_WAIT_TOLERANCE:
		fEndpointCurrentError := fEndpointTargetForce - fForce;
		IF ABS(fEndpointCurrentError) <= fEndpointTolerance OR
			(fEndpointStartError > 0.0 AND fEndpointCurrentError <= 0.0) OR
			(fEndpointStartError < 0.0 AND fEndpointCurrentError >= 0.0) THEN
			bExecuteVelMove := FALSE;
			stateHalt := TRUE;
			nVelocityState := 3;
			nSeqState := STATE_FORCE_WAIT_STOP;
		END_IF

	STATE_FORCE_WAIT_STOP:
		IF bHaltDone THEN
			stateHalt := FALSE;
			nVelocityState := 4;
			IF bZeroForceUnload THEN
				IF bSyncEnabled AND nEndpointSyncPoint <> SYNC_NONE THEN
					bForceEndpointReady := TRUE;
					nSyncPoint := nEndpointSyncPoint;
					nSyncCycle := nEndpointSyncCycle;
					nSeqState := STATE_FORCE_HOLD;
				ELSE
					bZeroForceUnload := FALSE;
					nSeqState := nAfterEndpointState;
				END_IF
			ELSE
				nVelocityUpdateCounter := VELOCITY_UPDATE_CYCLES;
				fLastSentVelocity := 0.0;
				nSeqState := STATE_FORCE_HOLD;
			END_IF
		END_IF

	STATE_FORCE_HOLD: // P-regulate while the timer runs and the peer catches up.
		IF bZeroForceUnload AND NOT bSyncRelease THEN
			// Wait at standstill for the other axis; never reload across zero.
			bExecuteVelMove := FALSE;
		ELSIF bForceEndpointReady AND bSyncRelease THEN
			bExecuteVelMove := FALSE;
			bForceEndpointReady := FALSE;
			bZeroForceUnload := FALSE;
			nSyncPoint := SYNC_NONE;
			nSyncCycle := 0;
			nEndpointSyncPoint := SYNC_NONE;
			IF nVelocityState = 4 THEN
				nSeqState := nAfterEndpointState;
			ELSE
				stateHalt := TRUE;
				nVelocityState := 3;
				nSeqState := STATE_FORCE_EXIT_WAIT_STOP;
			END_IF
		ELSE
			fForceError := fEndpointTargetForce - fForce;

			// Proportional correction begins only after the initial
			// constant-speed approach has reached the endpoint.
			fCmdVelocity := (fForceError * stSettings.fKp) *
				INT_TO_LREAL(FORCE_POLARITY);
			fCmdVelocity := LIMIT(
				-fForceRegMaxVelocity,
				fCmdVelocity,
				fForceRegMaxVelocity);
			fPendingVelocity := ABS(fCmdVelocity);
			IF fCmdVelocity >= 0.0 THEN
				mcPendingDirection := MC_Positive_Direction;
			ELSE
				mcPendingDirection := MC_Negative_Direction;
			END_IF
			IF nVelocityUpdateCounter < VELOCITY_UPDATE_CYCLES THEN
				nVelocityUpdateCounter := nVelocityUpdateCounter + 1;
			END_IF

			// Tiny corrections are replaced by a powered position hold.
			IF fPendingVelocity <= fForceRegMinVelocity THEN
				bExecuteVelMove := FALSE;
				IF nVelocityState <> 3 AND nVelocityState <> 4 THEN
					stateHalt := TRUE;
					nVelocityState := 3;
				ELSIF nVelocityState = 3 AND bHaltDone THEN
					stateHalt := FALSE;
					nVelocityState := 4;
				END_IF
			ELSIF nVelocityState = 3 THEN
				IF bHaltDone THEN
					stateHalt := FALSE;
					nVelocityState := 0;
				END_IF
			ELSIF nVelocityState = 4 THEN
				nVelocityState := 0;
			ELSIF nVelocityState = 2 THEN
				fCmdVelocity := fPendingVelocity;
				mcDirection := mcPendingDirection;
				IF mcDirection = MC_Positive_Direction THEN
					nLoadDirection := 1;
					nLastMotionDirection := 1;
				ELSE
					nLoadDirection := -1;
					nLastMotionDirection := -1;
				END_IF
				bExecuteVelMove := TRUE;
				fLastSentVelocity := fCmdVelocity;
				nVelocityUpdateCounter := 0;
				nVelocityState := 1;
			ELSE
				IF nVelocityState = 0 THEN
					fCmdVelocity := fPendingVelocity;
					mcDirection := mcPendingDirection;
					IF mcDirection = MC_Positive_Direction THEN
						nLoadDirection := 1;
						nLastMotionDirection := 1;
					ELSE
						nLoadDirection := -1;
						nLastMotionDirection := -1;
					END_IF
					bExecuteVelMove := TRUE;
					fLastSentVelocity := fCmdVelocity;
					nVelocityUpdateCounter := 0;
					nVelocityState := 1;
				ELSIF nVelocityUpdateCounter >=
					VELOCITY_UPDATE_CYCLES AND
					(ABS(fPendingVelocity - fLastSentVelocity) >=
						fForceRegMinVelocity OR
					 mcPendingDirection <> mcDirection) THEN
					bExecuteVelMove := FALSE;
					nVelocityState := 2;
				END_IF
			END_IF

			// Hold time is accumulated only inside tolerance. Excursions
			// pause it and withdraw readiness without resetting elapsed time.
			IF ABS(fForceError) <= fEndpointTolerance THEN
				IF NOT bForceEndpointReady THEN
					fForceHoldElapsed := fForceHoldElapsed + CYCLE_TIME;
					IF fForceHoldElapsed >= fEndpointHoldTime THEN
						IF bSyncEnabled AND
							nEndpointSyncPoint <> SYNC_NONE THEN
							// Publish barrier readiness only at confirmed
							// standstill. Otherwise both axes could be released
							// while one is still executing a correction.
							bExecuteVelMove := FALSE;
							IF nVelocityState = 4 THEN
								bForceEndpointReady := TRUE;
								nSyncPoint := nEndpointSyncPoint;
								nSyncCycle := nEndpointSyncCycle;
							ELSE
								stateHalt := TRUE;
								nVelocityState := 3;
								nSeqState :=
									STATE_FORCE_READY_WAIT_STOP;
							END_IF
						ELSE
							bExecuteVelMove := FALSE;
							IF nVelocityState = 4 THEN
								nSeqState := nAfterEndpointState;
							ELSE
								stateHalt := TRUE;
								nVelocityState := 3;
								nSeqState :=
									STATE_FORCE_EXIT_WAIT_STOP;
							END_IF
						END_IF
					END_IF
				END_IF
			ELSIF bForceEndpointReady THEN
				bForceEndpointReady := FALSE;
				nSyncPoint := SYNC_NONE;
				nSyncCycle := 0;
			END_IF
		END_IF

	STATE_FORCE_EXIT_WAIT_STOP:
		bExecuteVelMove := FALSE;
		IF bHaltDone THEN
			stateHalt := FALSE;
			nVelocityState := 4;
			nSeqState := nAfterEndpointState;
		END_IF

	STATE_FORCE_READY_WAIT_STOP:
		bExecuteVelMove := FALSE;
		IF bHaltDone THEN
			stateHalt := FALSE;
			nVelocityState := 4;
			fForceError := fEndpointTargetForce - fForce;
			IF ABS(fForceError) <= fEndpointTolerance THEN
				bForceEndpointReady := TRUE;
				nSyncPoint := nEndpointSyncPoint;
				nSyncCycle := nEndpointSyncCycle;
			END_IF
			nSeqState := STATE_FORCE_HOLD;
		END_IF
END_CASE
END_ACTION

ACTION mode1:

// =========================================================
//                  Mode 1: Maintained jog
// =========================================================

CASE nSeqState OF
	STATE_IDLE:
		IF stMoveCommand.bExecute THEN
			IF NOT ((stMoveCommand.fMoveVelocity =
				stMoveCommand.fMoveVelocity) AND
				ABS(stMoveCommand.fMoveVelocity) > 0.0 AND
				ABS(stMoveCommand.fMoveVelocity) < 1.0E300) THEN
				stMoveCommand.bExecute := FALSE;
				SetError(
					nCode := ERROR_INVALID_RUNTIME_VALUE,
					nNativeErrorID := 0,
					bRequestHalt := TRUE);
			ELSIF ABS(stMoveCommand.fMoveVelocity) >
				ABS(stSettings.fMaxVelocity) THEN
				stMoveCommand.bExecute := FALSE;
				SetError(
					nCode := ERROR_VELOCITY_LIMIT,
					nNativeErrorID := 0,
					bRequestHalt := TRUE);
			ELSE
				nSystemStatus := STATUS_BASIC_MOVE;
				fCmdVelocity := ABS(stMoveCommand.fMoveVelocity);
				IF stMoveCommand.fMoveVelocity > 0.0 THEN
					mcDirection := MC_Positive_Direction;
					nLastMotionDirection := 1;
				ELSE
					mcDirection := MC_Negative_Direction;
					nLastMotionDirection := -1;
				END_IF
				nLastJogLeaseCounter :=
					stMoveCommand.nJogLeaseCounter;
				bExecuteVelMove := TRUE;
				nSeqState := STATE_MODE_RUN;
			END_IF
		END_IF

	STATE_MODE_RUN:
		IF NOT stMoveCommand.bExecute THEN
			bExecuteVelMove := FALSE;
			stateHalt := TRUE;
			nSeqState := STATE_MODE_START;
		END_IF

	STATE_MODE_START:
		IF bHaltDone THEN
			stateHalt := FALSE;
			bOperationCompleted := TRUE;
			nSeqState := STATE_IDLE;
		END_IF
END_CASE
END_ACTION

ACTION mode2:


// =========================================================
//                  Mode 2: Constant Force
// =========================================================
// One PI-regulated target force for one duration.

CASE nSeqState OF
	STATE_IDLE: // Wait for command
		bExecuteVelMove := FALSE;
		fCmdVelocity := 0.0;
		fForceErrorIntegral := 0.0;
		fLastSentVelocity := 0.0;
		IF stMoveCommand.bExecute THEN
			stMoveCommand.bExecute := FALSE;
			nSystemStatus := STATUS_FORCE_MODE;
			nVelocityState := 0;
			nLoadDirection := 0;
			nLastMotionDirection := 0;
			nReliefSourceDirection := 0;
			nSeqState := STATE_MODE_START;
		END_IF

	STATE_MODE_START: // Initialize the single force/time command.
		fTargetForce := stMoveCommand.fTargetForce;
		fForceErrorIntegral := 0.0;
		fMode2HoldElapsed := 0.0;
		fLastSentVelocity := 0.0;
		nVelocityUpdateCounter := VELOCITY_UPDATE_CYCLES;
		nSeqState := STATE_MODE_RUN;

	STATE_MODE_RUN: // Force Regulation Loop (PI Regulator)
		fForceError := fTargetForce - fForce;
		
		fForceErrorIntegral := fForceErrorIntegral + (fForceError * CYCLE_TIME);
		fForceErrorIntegral := LIMIT(-stSettings.fIntegralLimit, fForceErrorIntegral, stSettings.fIntegralLimit);
		
		// Apply the fixed machine force polarity to the PI output.
		fCmdVelocity := ((fForceError * stSettings.fKp) +
			(fForceErrorIntegral * stSettings.fKi)) *
			INT_TO_LREAL(FORCE_POLARITY);
		fCmdVelocity := LIMIT(-stSettings.fMaxVelocity, fCmdVelocity, stSettings.fMaxVelocity);
		
		IF nVelocityUpdateCounter < VELOCITY_UPDATE_CYCLES THEN
			nVelocityUpdateCounter := nVelocityUpdateCounter + 1;
		END_IF

		IF ABS(fForceError) <= stSettings.fForceTolerance THEN
			// Stop in the force deadband without powering the axis off.
			bExecuteVelMove := FALSE;
			IF nVelocityState <> 3 AND nVelocityState <> 4 THEN
				stateHalt := TRUE;
				nVelocityState := 3;
			ELSIF nVelocityState = 3 AND bHaltDone THEN
				stateHalt := FALSE;
				nVelocityState := 4;
			END_IF
		ELSIF nVelocityState = 3 THEN
			IF bHaltDone THEN
				stateHalt := FALSE;
				nVelocityState := 0;
			END_IF
		ELSIF nVelocityState = 4 THEN
			// The axis is stopped and the force left the deadband.
			nVelocityState := 0;
		ELSIF nVelocityState = 2 THEN
			fCmdVelocity := fPendingVelocity;
			mcDirection := mcPendingDirection;
			bExecuteVelMove := TRUE;
			fLastSentVelocity := fCmdVelocity;
			nVelocityUpdateCounter := 0;
			nVelocityState := 1;
		ELSE
			IF fCmdVelocity >= 0.0 THEN
				mcPendingDirection := MC_Positive_Direction;
			ELSE
				mcPendingDirection := MC_Negative_Direction;
			END_IF
			fPendingVelocity := ABS(fCmdVelocity);

			IF nVelocityState = 0 THEN
				fCmdVelocity := fPendingVelocity;
				mcDirection := mcPendingDirection;
				bExecuteVelMove := TRUE;
				fLastSentVelocity := fCmdVelocity;
				nVelocityUpdateCounter := 0;
				nVelocityState := 1;
			ELSIF nVelocityUpdateCounter >= VELOCITY_UPDATE_CYCLES AND
				(ABS(fPendingVelocity - fLastSentVelocity) >= VELOCITY_UPDATE_DELTA OR
				 mcPendingDirection <> mcDirection) THEN
				bExecuteVelMove := FALSE;
				nVelocityState := 2;
			END_IF
		END_IF
		
		// Count only time spent stopped inside the force tolerance. Leaving the
		// deadband pauses this accumulated time; re-entry resumes it.
		IF ABS(fForceError) <= stSettings.fForceTolerance AND
			nVelocityState = 4 THEN
			fMode2HoldElapsed := fMode2HoldElapsed + CYCLE_TIME;
			IF fMode2HoldElapsed >= stMoveCommand.fForceDuration THEN
				bExecuteVelMove := FALSE;
				stateHalt := FALSE;
				nVelocityState := 0;
				bOperationCompleted := TRUE;
				nSeqState := STATE_IDLE;
			END_IF
		END_IF
END_CASE
END_ACTION

ACTION positionEndpoint:

CASE nSeqState OF
	STATE_POSITION_PREPARE:
		fbMC_MoveRelative1.Execute := FALSE;
		fPositionHoldElapsed := 0.0;
		IF ABS(fTargetDist1) <= POSITION_EPSILON THEN
			// No movement is needed, but a configured Mode 3 hold still applies.
			IF fEndpointHoldTime > 0.0 THEN
				nSeqState := STATE_POSITION_HOLD;
			ELSIF bSyncEnabled AND nEndpointSyncPoint <> SYNC_NONE THEN
				nSyncPoint := nEndpointSyncPoint;
				nSyncCycle := nEndpointSyncCycle;
				nSeqState := STATE_POSITION_BARRIER;
			ELSE
				nSeqState := nAfterEndpointState;
			END_IF
		ELSE
			IF fTargetDist1 > 0.0 THEN
				nLastMotionDirection := 1;
			ELSE
				nLastMotionDirection := -1;
			END_IF
			nSeqState := STATE_POSITION_EXECUTE;
		END_IF

	STATE_POSITION_EXECUTE: // One scan with Execute low before reuse.
		fbMC_MoveRelative1.Execute := TRUE;
		nSeqState := STATE_POSITION_WAIT;

	STATE_POSITION_WAIT:
		IF fbMC_MoveRelative1.Done THEN
			fbMC_MoveRelative1.Execute := FALSE;
			IF fEndpointHoldTime > 0.0 THEN
				nSeqState := STATE_POSITION_HOLD;
			ELSIF bSyncEnabled AND nEndpointSyncPoint <> SYNC_NONE THEN
				nSyncPoint := nEndpointSyncPoint;
				nSyncCycle := nEndpointSyncCycle;
				nSeqState := STATE_POSITION_BARRIER;
			ELSE
				nSeqState := nAfterEndpointState;
			END_IF
		END_IF

	STATE_POSITION_HOLD: // Powered NC loop holds for the endpoint duration.
		fPositionHoldElapsed := fPositionHoldElapsed + CYCLE_TIME;
		IF fPositionHoldElapsed >= fEndpointHoldTime THEN
			IF bSyncEnabled AND nEndpointSyncPoint <> SYNC_NONE THEN
				nSyncPoint := nEndpointSyncPoint;
				nSyncCycle := nEndpointSyncCycle;
				nSeqState := STATE_POSITION_BARRIER;
			ELSE
				nSeqState := nAfterEndpointState;
			END_IF
		END_IF

	STATE_POSITION_BARRIER: // Powered NC loop holds while peer catches up.
		nSyncPoint := nEndpointSyncPoint;
		nSyncCycle := nEndpointSyncCycle;
		IF NOT bSyncEnabled OR bSyncRelease THEN
			nSyncPoint := SYNC_NONE;
			nSyncCycle := 0;
			nEndpointSyncPoint := SYNC_NONE;
			nSeqState := nAfterEndpointState;
		END_IF
END_CASE
END_ACTION

METHOD PrepareForceEndpoint
VAR_INPUT
	fTargetForceValue : LREAL;
	fRate             : LREAL;
	fTolerance        : LREAL;
	fHoldTime         : LREAL;
	nTargetSyncPoint  : BYTE;
	nTargetSyncCycle  : INT;
	nNextState        : INT;
END_VAR

fEndpointTargetForce := fTargetForceValue;
fEndpointRate := ABS(fRate);
fEndpointTolerance := fTolerance;
fEndpointHoldTime := fHoldTime;
bZeroForceUnload := FALSE;
nEndpointSyncPoint := nTargetSyncPoint;
nEndpointSyncCycle := nTargetSyncCycle;
nAfterEndpointState := nNextState;
nSeqState := STATE_FORCE_PREPARE;
END_METHOD

METHOD PreparePositionEndpoint
VAR_INPUT
	fTargetPosition : LREAL;
	fRate           : LREAL;
	fHoldTime       : LREAL;
	nTargetSyncPoint: BYTE;
	nTargetSyncCycle: INT;
	nNextState      : INT;
END_VAR

fEndpointTargetPosition := fTargetPosition;
fTargetDist1 := fEndpointTargetPosition - fActPosition;
fTargetVel1 := ABS(fRate);
fEndpointHoldTime := fHoldTime;
nEndpointSyncPoint := nTargetSyncPoint;
nEndpointSyncCycle := nTargetSyncCycle;
nAfterEndpointState := nNextState;
nSeqState := STATE_POSITION_PREPARE;
END_METHOD

METHOD SetError
VAR_INPUT
	nCode          : UDINT;
	nNativeErrorID : UDINT;
	bRequestHalt   : BOOL;
END_VAR

bError := TRUE;
nErrorCode := nCode;
nAxisErrorID := nNativeErrorID;
ClearActiveCommand();
IF bRequestHalt THEN
	stateHalt := TRUE;
	nSeqState := STATE_ERROR_STOPPING;
ELSE
	stateHalt := FALSE;
	nSeqState := STATE_ERROR_LATCHED;
END_IF
END_METHOD

ACTION testSequence:

// Shared pre-test, main-test and post-test sequence for mode 3.
// All stored coordinates are references only; every position command is relative.

// Criterion 2 ends a single test immediately when its signed level is crossed.
IF bSinglePrimaryActive AND stMoveCommand.nStop2Mode > 0 THEN
	bSingleStopReached := FALSE;
	IF stMoveCommand.nStop2Mode = 1 THEN
		fStop2CurrentError := fStop2TargetPosition - fActPosition;
		IF ABS(fStop2CurrentError) <= POSITION_EPSILON OR
			(fStop2StartError > 0.0 AND fStop2CurrentError <= 0.0) OR
			(fStop2StartError < 0.0 AND fStop2CurrentError >= 0.0) THEN
			bSingleStopReached := TRUE;
		END_IF
	ELSIF stMoveCommand.nStop2Mode = 2 THEN
		fStop2CurrentError := stMoveCommand.fStop2Value - fForce;
		IF ABS(fStop2CurrentError) <=
			SEL(stMoveCommand.fSingleForceTolerance < 0.0,
				stMoveCommand.fSingleForceTolerance,
				MAX(ABS(stMoveCommand.fStop2Value) *
					ABS(stMoveCommand.fSingleForceTolerance) / 100.0,
					stSettings.fForceTolerance)) OR
			(fStop2StartError > 0.0 AND fStop2CurrentError <= 0.0) OR
			(fStop2StartError < 0.0 AND fStop2CurrentError >= 0.0) THEN
			bSingleStopReached := TRUE;
		END_IF
	ELSIF stMoveCommand.nStop2Mode = 3 THEN
		IF NOT bSingleRuptureArmed AND
			ABS(fForce) >= fSingleStartForce + stSettings.fForceTolerance THEN
			bSingleRuptureArmed := TRUE;
		END_IF
		IF bSingleRuptureArmed THEN
			fSinglePeakForce := MAX(fSinglePeakForce, ABS(fForce));
		END_IF
		IF bSingleRuptureArmed AND ABS(fForce) <= fSinglePeakForce *
			(1.0 - stMoveCommand.fStop2Value / 100.0) THEN
			bSingleStopReached := TRUE;
		END_IF
	END_IF

	IF bSingleStopReached THEN
		fbMC_MoveRelative1.Execute := FALSE;
		bExecuteVelMove := FALSE;
		bSinglePrimaryActive := FALSE;
		stateHalt := TRUE;
		nSeqState := STATE_SINGLE_WAIT_STOP;
	END_IF
END_IF

CASE nSeqState OF
	STATE_IDLE: // Start a test. MATLAB keeps command values unchanged while bWorking is TRUE.
		fbMC_MoveRelative1.Execute := FALSE;
		bExecuteVelMove := FALSE;
		stateHalt := FALSE;
		bSinglePrimaryActive := FALSE;
		bForceEndpointReady := FALSE;
		nSyncPoint := SYNC_NONE;
		nSyncCycle := 0;
		nEndpointSyncPoint := SYNC_NONE;
		nEndpointSyncCycle := 0;

		IF stMoveCommand.bExecute THEN
			stMoveCommand.bExecute := FALSE;
			IF (stMoveCommand.bIncludePreTest AND
				(stMoveCommand.bPreloadEnabled OR
				 stMoveCommand.nPreCycleCount > 0) AND
				(NOT ((stMoveCommand.fPreTestRate =
					stMoveCommand.fPreTestRate) AND
					ABS(stMoveCommand.fPreTestRate) > 0.0 AND
					ABS(stMoveCommand.fPreTestRate) < 1.0E300) OR
				 ABS(stMoveCommand.fPreTestRate) >
					ABS(stSettings.fMaxVelocity))) OR
				(NOT stMoveCommand.bPreTestOnly AND
				 (NOT ((stMoveCommand.fTestRate =
					stMoveCommand.fTestRate) AND
					ABS(stMoveCommand.fTestRate) > 0.0 AND
					ABS(stMoveCommand.fTestRate) < 1.0E300) OR
				  ABS(stMoveCommand.fTestRate) >
					ABS(stSettings.fMaxVelocity))) THEN
				SetError(
					nCode := ERROR_VELOCITY_LIMIT,
					nNativeErrorID := 0,
					bRequestHalt := TRUE);
			ELSIF stMoveCommand.nCycleCount < 0 OR
				stMoveCommand.nCycleCount > 50 OR
				stMoveCommand.nPreCycleCount < 0 OR
				stMoveCommand.nPreCycleCount > 50 OR
				(stMoveCommand.bPreTestOnly AND NOT stMoveCommand.bIncludePreTest) OR
				NOT ((stMoveCommand.fPreTestForceTolerance = stMoveCommand.fPreTestForceTolerance) AND
					ABS(stMoveCommand.fPreTestForceTolerance) < 1.0E300 AND
					stMoveCommand.fPreTestForceTolerance >= -100.0) OR
				NOT ((stMoveCommand.fPreloadHoldTime = stMoveCommand.fPreloadHoldTime) AND
					ABS(stMoveCommand.fPreloadHoldTime) < 1.0E300 AND
					stMoveCommand.fPreloadHoldTime >= 0.0) OR
				NOT ((stMoveCommand.fPreCycleHoldTime = stMoveCommand.fPreCycleHoldTime) AND
					ABS(stMoveCommand.fPreCycleHoldTime) < 1.0E300 AND
					stMoveCommand.fPreCycleHoldTime >= 0.0) OR
				NOT ((stMoveCommand.fSingleForceTolerance = stMoveCommand.fSingleForceTolerance) AND
					ABS(stMoveCommand.fSingleForceTolerance) < 1.0E300 AND
					stMoveCommand.fSingleForceTolerance >= -100.0) OR
				NOT ((stMoveCommand.fSingleForceHoldTime = stMoveCommand.fSingleForceHoldTime) AND
					ABS(stMoveCommand.fSingleForceHoldTime) < 1.0E300 AND
					stMoveCommand.fSingleForceHoldTime >= 0.0) OR
				NOT ((stMoveCommand.fCyclicForceTolerance = stMoveCommand.fCyclicForceTolerance) AND
					ABS(stMoveCommand.fCyclicForceTolerance) < 1.0E300 AND
					stMoveCommand.fCyclicForceTolerance >= -100.0) OR
				NOT ((stMoveCommand.fCyclicForceHoldTime = stMoveCommand.fCyclicForceHoldTime) AND
					ABS(stMoveCommand.fCyclicForceHoldTime) < 1.0E300 AND
					stMoveCommand.fCyclicForceHoldTime >= 0.0) OR
				(stMoveCommand.nStop2Mode = 3 AND
					stSettings.fForceTolerance <= 0.0) THEN
				bError := TRUE;
				nErrorCode := ERROR_INVALID_CONFIGURATION;
				stateHalt := TRUE;
				nSeqState := STATE_ERROR_STOPPING;
			ELSE
				fTestStartPos := fActPosition;
				fPreTestFinalPos := fTestStartPos;
				nCurrentCycle := 1;
				nCurrentPreCycle := 1;
				nLoadDirection := 0;
				nLastMotionDirection := 0;
				nReliefSourceDirection := 0;
				nVelocityState := 0;

				IF stMoveCommand.bIncludePreTest THEN
					IF stMoveCommand.bPreloadEnabled THEN
						nSystemStatus := STATUS_PRETENSION;
					ELSE
						nSystemStatus := STATUS_PRETEST_CYCLIC;
					END_IF
					nSeqState := STATE_PRELOAD;
				ELSE
					IF stMoveCommand.nCycleCount > 0 THEN
						nSystemStatus := STATUS_CYCLIC_TEST;
					ELSE
						nSystemStatus := STATUS_SINGLE_TEST;
					END_IF
					nSeqState := STATE_SELECT_MAIN_TEST;
				END_IF
			END_IF
		END_IF

	STATE_PRELOAD: // Optional one-time force preload.
		nCurrentPreCycle := 1;
		IF stMoveCommand.bPreloadEnabled THEN
			nSystemStatus := STATUS_PRETENSION;
			fEndpointTargetForce := stMoveCommand.fPreloadValue;
			fEndpointRate := ABS(stMoveCommand.fPreTestRate);
			fEndpointTolerance := SEL(stMoveCommand.fPreTestForceTolerance < 0.0,
				stMoveCommand.fPreTestForceTolerance,
				MAX(ABS(fEndpointTargetForce) *
					ABS(stMoveCommand.fPreTestForceTolerance) / 100.0,
					stSettings.fForceTolerance));
			fEndpointHoldTime := stMoveCommand.fPreloadHoldTime;
			nEndpointSyncPoint := SYNC_PRETENSION_DONE;
			nEndpointSyncCycle := 0;
			nAfterEndpointState := STATE_CAPTURE_TEST_START;
			nSeqState := STATE_FORCE_PREPARE;
		ELSE
			nSystemStatus := STATUS_PRETEST_CYCLIC;
			nSeqState := STATE_PRE_CYCLE_LOAD;
		END_IF

	STATE_CAPTURE_TEST_START: // Capture post-pretension test start.
		fTestStartPos := fActPosition;
		IF stMoveCommand.nPreCycleCount > 0 THEN
			nSystemStatus := STATUS_PRETEST_CYCLIC;
			nSeqState := STATE_PRE_CYCLE_LOAD;
		ELSE
			nSeqState := STATE_CAPTURE_PRETEST_FINAL;
		END_IF

	STATE_PRE_CYCLE_LOAD: // Pre-conditioning force-load endpoint.
		nSystemStatus := STATUS_PRETEST_CYCLIC;
		IF nCurrentPreCycle > stMoveCommand.nPreCycleCount THEN
			nSeqState := STATE_PRETEST_BARRIER;
		ELSE
			fEndpointTargetForce := stMoveCommand.fPreCycleLoadValue;
			fEndpointRate := ABS(stMoveCommand.fPreTestRate);
			fEndpointTolerance := SEL(stMoveCommand.fPreTestForceTolerance < 0.0,
				stMoveCommand.fPreTestForceTolerance,
				MAX(ABS(fEndpointTargetForce) *
					ABS(stMoveCommand.fPreTestForceTolerance) / 100.0,
					stSettings.fForceTolerance));
			fEndpointHoldTime := stMoveCommand.fPreCycleHoldTime;
			nEndpointSyncPoint := SYNC_LOAD_DONE;
			nEndpointSyncCycle := nCurrentPreCycle;
			nAfterEndpointState := STATE_PRE_CYCLE_UNLOAD;
			nSeqState := STATE_FORCE_PREPARE;
		END_IF

	STATE_PRE_CYCLE_UNLOAD: // Force unload or return to test start.
		nSystemStatus := STATUS_PRETEST_CYCLIC;
		IF stMoveCommand.bPreUnloadToStart THEN
			fEndpointTargetPosition := fTestStartPos;
			fTargetDist1 := fEndpointTargetPosition - fActPosition;
			fTargetVel1 := ABS(stMoveCommand.fPreTestRate);
			fEndpointHoldTime := stMoveCommand.fPreCycleHoldTime;
			IF nCurrentPreCycle = stMoveCommand.nPreCycleCount THEN
				nEndpointSyncPoint := SYNC_PRETEST_DONE;
				nAfterEndpointState := STATE_CAPTURE_PRETEST_FINAL;
			ELSE
				nEndpointSyncPoint := SYNC_UNLOAD_DONE;
				nAfterEndpointState := STATE_PRE_CYCLE_NEXT;
			END_IF
			nEndpointSyncCycle := nCurrentPreCycle;
			nSeqState := STATE_POSITION_PREPARE;
		ELSE
			fEndpointTargetForce := stMoveCommand.fPreUnloadValue;
			fEndpointRate := ABS(stMoveCommand.fPreTestRate);
			fEndpointTolerance := SEL(stMoveCommand.fPreTestForceTolerance < 0.0,
				stMoveCommand.fPreTestForceTolerance,
				MAX(ABS(fEndpointTargetForce) *
					ABS(stMoveCommand.fPreTestForceTolerance) / 100.0,
					stSettings.fForceTolerance));
			fEndpointHoldTime := stMoveCommand.fPreCycleHoldTime;
			IF nCurrentPreCycle = stMoveCommand.nPreCycleCount THEN
				nEndpointSyncPoint := SYNC_PRETEST_DONE;
				nAfterEndpointState := STATE_CAPTURE_PRETEST_FINAL;
			ELSE
				nEndpointSyncPoint := SYNC_UNLOAD_DONE;
				nAfterEndpointState := STATE_PRE_CYCLE_NEXT;
			END_IF
			nEndpointSyncCycle := nCurrentPreCycle;
			nSeqState := STATE_FORCE_PREPARE;
		END_IF

	STATE_PRE_CYCLE_NEXT:
		nCurrentPreCycle := nCurrentPreCycle + 1;
		nSeqState := STATE_PRE_CYCLE_LOAD;

	STATE_CAPTURE_PRETEST_FINAL: // Final pre-test endpoint passed its barrier.
		fPreTestFinalPos := fActPosition;
		IF stMoveCommand.bPreTestOnly THEN
			nSystemStatus := STATUS_POSTTEST;
			nSeqState := STATE_POSTTEST_SELECT;
		ELSE
			IF stMoveCommand.nCycleCount > 0 THEN
				nSystemStatus := STATUS_CYCLIC_TEST;
			ELSE
				nSystemStatus := STATUS_SINGLE_TEST;
			END_IF
			nSeqState := STATE_SELECT_MAIN_TEST;
		END_IF

	STATE_PRETEST_BARRIER: // No final endpoint; explicit pre-test barrier.
		nSystemStatus := STATUS_PRETEST_CYCLIC;
		nSyncPoint := SYNC_PRETEST_DONE;
		nSyncCycle := 0;
		IF NOT bSyncEnabled OR bSyncRelease THEN
			nSyncPoint := SYNC_NONE;
			fPreTestFinalPos := fActPosition;
			IF stMoveCommand.bPreTestOnly THEN
				nSystemStatus := STATUS_POSTTEST;
				nSeqState := STATE_POSTTEST_SELECT;
			ELSE
				IF stMoveCommand.nCycleCount > 0 THEN
					nSystemStatus := STATUS_CYCLIC_TEST;
				ELSE
					nSystemStatus := STATUS_SINGLE_TEST;
				END_IF
				nSeqState := STATE_SELECT_MAIN_TEST;
			END_IF
		END_IF

	STATE_SELECT_MAIN_TEST: // Positive cycle count selects cyclic.
		IF stMoveCommand.nCycleCount > 0 THEN
			nSystemStatus := STATUS_CYCLIC_TEST;
			nSeqState := STATE_CYCLIC_LOAD;
		ELSE
			nSystemStatus := STATUS_SINGLE_TEST;
			nSeqState := STATE_SINGLE_START;
		END_IF

	// -----------------------------------------------------
	// Mode 3: cyclic load endpoint followed by unload endpoint
	// -----------------------------------------------------
	STATE_CYCLIC_LOAD:
		nSystemStatus := STATUS_CYCLIC_TEST;
		IF nCurrentCycle > stMoveCommand.nCycleCount THEN
			nSeqState := STATE_POSTTEST_SELECT;
		ELSIF stMoveCommand.nLoadMode = 1 THEN
			fEndpointTargetPosition := fPreTestFinalPos +
				stMoveCommand.fLoadValues[nCurrentCycle];
			fTargetDist1 := fEndpointTargetPosition - fActPosition;
			fTargetVel1 := ABS(stMoveCommand.fTestRate);
			fEndpointHoldTime := stMoveCommand.fCyclicForceHoldTime;
			IF fTargetDist1 > POSITION_EPSILON THEN
				nLoadDirection := 1;
			ELSIF fTargetDist1 < -POSITION_EPSILON THEN
				nLoadDirection := -1;
			END_IF
			nEndpointSyncPoint := SYNC_LOAD_DONE;
			nEndpointSyncCycle := nCurrentCycle;
			nAfterEndpointState := STATE_CYCLIC_UNLOAD;
			nSeqState := STATE_POSITION_PREPARE;
		ELSIF stMoveCommand.nLoadMode = 2 THEN
			fEndpointTargetForce := stMoveCommand.fLoadValues[nCurrentCycle];
			fEndpointRate := ABS(stMoveCommand.fTestRate);
			fEndpointTolerance := SEL(stMoveCommand.fCyclicForceTolerance < 0.0,
				stMoveCommand.fCyclicForceTolerance,
				MAX(ABS(fEndpointTargetForce) *
					ABS(stMoveCommand.fCyclicForceTolerance) / 100.0,
					stSettings.fForceTolerance));
			fEndpointHoldTime := stMoveCommand.fCyclicForceHoldTime;
			nEndpointSyncPoint := SYNC_LOAD_DONE;
			nEndpointSyncCycle := nCurrentCycle;
			nAfterEndpointState := STATE_CYCLIC_UNLOAD;
			nSeqState := STATE_FORCE_PREPARE;
		ELSE
			bError := TRUE;
			nErrorCode := ERROR_UNSUPPORTED_ENDPOINT;
			stateHalt := TRUE;
			nSeqState := STATE_ERROR_STOPPING;
		END_IF

	STATE_CYCLIC_UNLOAD:
		nSystemStatus := STATUS_CYCLIC_TEST;
		IF stMoveCommand.nUnloadMode = 1 THEN
			fEndpointTargetPosition := fPreTestFinalPos +
				stMoveCommand.fUnloadValues[nCurrentCycle];
			fTargetDist1 := fEndpointTargetPosition - fActPosition;
			fTargetVel1 := ABS(stMoveCommand.fTestRate);
			fEndpointHoldTime := stMoveCommand.fCyclicForceHoldTime;
			IF nCurrentCycle = stMoveCommand.nCycleCount THEN
				nEndpointSyncPoint := SYNC_MAIN_DONE;
				nAfterEndpointState := STATE_CYCLIC_COMPLETE;
			ELSE
				nEndpointSyncPoint := SYNC_UNLOAD_DONE;
				nAfterEndpointState := STATE_CYCLIC_NEXT;
			END_IF
			nEndpointSyncCycle := nCurrentCycle;
			nSeqState := STATE_POSITION_PREPARE;
		ELSIF stMoveCommand.nUnloadMode = 2 THEN
			fEndpointTargetForce := stMoveCommand.fUnloadValues[nCurrentCycle];
			fEndpointRate := ABS(stMoveCommand.fTestRate);
			fEndpointTolerance := SEL(stMoveCommand.fCyclicForceTolerance < 0.0,
				stMoveCommand.fCyclicForceTolerance,
				MAX(ABS(fEndpointTargetForce) *
					ABS(stMoveCommand.fCyclicForceTolerance) / 100.0,
					stSettings.fForceTolerance));
			fEndpointHoldTime := stMoveCommand.fCyclicForceHoldTime;
			IF nCurrentCycle = stMoveCommand.nCycleCount THEN
				nEndpointSyncPoint := SYNC_MAIN_DONE;
				nAfterEndpointState := STATE_CYCLIC_COMPLETE;
			ELSE
				nEndpointSyncPoint := SYNC_UNLOAD_DONE;
				nAfterEndpointState := STATE_CYCLIC_NEXT;
			END_IF
			nEndpointSyncCycle := nCurrentCycle;
			nSeqState := STATE_FORCE_PREPARE;
		ELSE
			bError := TRUE;
			nErrorCode := ERROR_UNSUPPORTED_ENDPOINT;
			stateHalt := TRUE;
			nSeqState := STATE_ERROR_STOPPING;
		END_IF

	STATE_CYCLIC_NEXT:
		nCurrentCycle := nCurrentCycle + 1;
		nSeqState := STATE_CYCLIC_LOAD;

	STATE_CYCLIC_COMPLETE: // Final unload also serves as main barrier.
		nCurrentCycle := nCurrentCycle + 1;
		nSeqState := STATE_POSTTEST_SELECT;

	// -----------------------------------------------------
	// Mode 3 single test: criterion 1 is the primary endpoint
	// -----------------------------------------------------
	STATE_SINGLE_START:
		nSystemStatus := STATUS_SINGLE_TEST;
		bSingleStopReached := FALSE;
		bSinglePrimaryActive := TRUE;
		fSingleStartForce := ABS(fForce);
		fSinglePeakForce := fSingleStartForce;
		bSingleRuptureArmed := FALSE;

		IF stMoveCommand.nStop2Mode = 1 THEN
			fStop2TargetPosition := fPreTestFinalPos + stMoveCommand.fStop2Value;
			fStop2StartError := fStop2TargetPosition - fActPosition;
		ELSIF stMoveCommand.nStop2Mode = 2 THEN
			fStop2StartError := stMoveCommand.fStop2Value - fForce;
		END_IF

		IF stMoveCommand.nStop1Mode = 1 THEN
			fEndpointTargetPosition := fPreTestFinalPos + stMoveCommand.fStop1Value;
			fTargetDist1 := fEndpointTargetPosition - fActPosition;
			fTargetVel1 := ABS(stMoveCommand.fTestRate);
			fEndpointHoldTime := stMoveCommand.fSingleForceHoldTime;
			IF fTargetDist1 > POSITION_EPSILON THEN
				nLoadDirection := 1;
			ELSIF fTargetDist1 < -POSITION_EPSILON THEN
				nLoadDirection := -1;
			END_IF
			nEndpointSyncPoint := SYNC_MAIN_DONE;
			nEndpointSyncCycle := 0;
			nAfterEndpointState := STATE_POSTTEST_SELECT;
			nSeqState := STATE_POSITION_PREPARE;
		ELSIF stMoveCommand.nStop1Mode = 2 THEN
			fEndpointTargetForce := stMoveCommand.fStop1Value;
			fEndpointRate := ABS(stMoveCommand.fTestRate);
			fEndpointTolerance := SEL(stMoveCommand.fSingleForceTolerance < 0.0,
				stMoveCommand.fSingleForceTolerance,
				MAX(ABS(fEndpointTargetForce) *
					ABS(stMoveCommand.fSingleForceTolerance) / 100.0,
					stSettings.fForceTolerance));
			fEndpointHoldTime := stMoveCommand.fSingleForceHoldTime;
			nEndpointSyncPoint := SYNC_MAIN_DONE;
			nEndpointSyncCycle := 0;
			nAfterEndpointState := STATE_POSTTEST_SELECT;
			nSeqState := STATE_FORCE_PREPARE;
		ELSE
			bSinglePrimaryActive := FALSE;
			bError := TRUE;
			nErrorCode := ERROR_UNSUPPORTED_ENDPOINT;
			stateHalt := TRUE;
			nSeqState := STATE_ERROR_STOPPING;
		END_IF

	STATE_SINGLE_WAIT_STOP: // Optional OR criterion stopped primary.
		IF bHaltDone THEN
			stateHalt := FALSE;
			nVelocityState := 0;
			nSeqState := STATE_SECONDARY_BARRIER;
		END_IF

	STATE_SECONDARY_BARRIER: // Secondary criterion ended test early.
		nSystemStatus := STATUS_SINGLE_TEST;
		nSyncPoint := SYNC_MAIN_DONE;
		nSyncCycle := 0;
		IF NOT bSyncEnabled OR bSyncRelease THEN
			nSyncPoint := SYNC_NONE;
			nSeqState := STATE_POSTTEST_SELECT;
		END_IF

	// -----------------------------------------------------
	// Post-test; reached only after normal main-test completion
	// -----------------------------------------------------
	STATE_POSTTEST_SELECT:
		nSystemStatus := STATUS_POSTTEST;
		bSinglePrimaryActive := FALSE;
		CASE stMoveCommand.nPostTestMode OF
			0: // Stay at the current position.
				fbMC_MoveRelative1.Execute := FALSE;
				bExecuteVelMove := FALSE;
				stateHalt := TRUE;
				nSeqState := STATE_POSTTEST_WAIT_STOP;

			1: // Return to the separately saved coordinate.
				IF bReferenceValid AND bSavedPositionValid THEN
					PreparePositionEndpoint(
						fTargetPosition := fSavedPosition,
						fRate := stMoveCommand.fTestRate,
						fHoldTime := 0.0,
						nTargetSyncPoint := SYNC_POSTTEST_DONE,
						nTargetSyncCycle := 0,
						nNextState := STATE_OPERATION_COMPLETE);
				ELSE
					stMoveCommand.bExecute := FALSE;
					SetError(
						nCode := ERROR_SAVED_POSITION_UNAVAILABLE,
						nNativeErrorID := 0,
						bRequestHalt := TRUE);
				END_IF

			2: // Return to the test-start position captured after pretension.
				PreparePositionEndpoint(
					fTargetPosition := fTestStartPos,
					fRate := stMoveCommand.fTestRate,
					fHoldTime := 0.0,
					nTargetSyncPoint := SYNC_POSTTEST_DONE,
					nTargetSyncCycle := 0,
					nNextState := STATE_OPERATION_COMPLETE);

			3: // Return to the actual position reached after pre-test.
				PreparePositionEndpoint(
					fTargetPosition := fPreTestFinalPos,
					fRate := stMoveCommand.fTestRate,
					fHoldTime := 0.0,
					nTargetSyncPoint := SYNC_POSTTEST_DONE,
					nTargetSyncCycle := 0,
					nNextState := STATE_OPERATION_COMPLETE);

			4: // Unload to zero tolerance without regulating back across zero.
				PrepareForceEndpoint(
					fTargetForceValue := 0.0,
					fRate := stMoveCommand.fTestRate,
					fTolerance := stSettings.fForceTolerance,
					fHoldTime := 0.0,
					nTargetSyncPoint := SYNC_POSTTEST_DONE,
					nTargetSyncCycle := 0,
					nNextState := STATE_OPERATION_COMPLETE);
				bZeroForceUnload := TRUE;

		ELSE
			stMoveCommand.bExecute := FALSE;
			SetError(
				nCode := ERROR_UNSUPPORTED_POST_ACTION,
				nNativeErrorID := 0,
				bRequestHalt := TRUE);
		END_CASE

	STATE_POSTTEST_WAIT_STOP:
		IF bHaltDone THEN
			stateHalt := FALSE;
			nSeqState := STATE_POSTTEST_BARRIER;
		END_IF

	STATE_POSTTEST_BARRIER: // Stay mode participates in post-test barrier.
		nSystemStatus := STATUS_POSTTEST;
		nSyncPoint := SYNC_POSTTEST_DONE;
		nSyncCycle := 0;
		IF NOT bSyncEnabled OR bSyncRelease THEN
			nSyncPoint := SYNC_NONE;
			nSeqState := STATE_OPERATION_COMPLETE;
		END_IF

	STATE_OPERATION_COMPLETE:
		nSystemStatus := STATUS_IDLE;
		nSyncPoint := SYNC_NONE;
		nSyncCycle := 0;
		bOperationCompleted := TRUE;
		nSeqState := STATE_IDLE;

	STATE_RESTORE_COMPLETE: // Standalone saved-position restore completed.
		nSystemStatus := STATUS_IDLE;
		bOperationCompleted := TRUE;
		nSeqState := STATE_IDLE;
END_CASE
END_ACTION

END_FUNCTION_BLOCK

// ---- POUs/fb_AxisStatusPublisher.TcPOU
FUNCTION_BLOCK fb_AxisStatusPublisher
VAR_INPUT
	fActPosition       : LREAL;
	bPowerStatus       : BOOL;
	bHoming            : BOOL;
	bHomed             : BOOL;
	bStopped           : BOOL;
	bProtectiveStop    : BOOL;
	bControllerHalt    : BOOL; // TRUE for PLC-owned regulation/sequence halt
	bSafetyError       : BOOL;
	nSafetyErrorCode   : UDINT;
	nSafetyAxisErrorID : UDINT;
	bMovementBusy      : BOOL;
	bMovementError     : BOOL;
	nMovementStatus    : INT;
	nMovementErrorCode : UDINT;
	nMovementAxisErrorID : UDINT;
	nOperationCounter  : UDINT;
	bSavedPositionValid: BOOL;
	bStartError        : BOOL;
	nStartErrorCode    : UDINT;
END_VAR

VAR_IN_OUT
	stSystemStatus : ST_SystemStatus;
END_VAR

VAR CONSTANT
	INTERFACE_VERSION : UDINT := 7;
END_VAR


stSystemStatus.fActPosition := 50.0 - fActPosition;
stSystemStatus.bPowered := bPowerStatus;
stSystemStatus.bHoming := bHoming;
stSystemStatus.bHomed := bHomed;
stSystemStatus.bStopped := bStopped;
stSystemStatus.bWorking := bMovementBusy OR bHoming OR
	bProtectiveStop OR stSystemStatus.bTarWorking;
stSystemStatus.nOperationCounter := nOperationCounter;
stSystemStatus.nInterfaceVersion := INTERFACE_VERSION;
stSystemStatus.bSavedPositionValid := bSavedPositionValid;
stSystemStatus.bError := bMovementError OR bSafetyError OR bStartError;

IF stSystemStatus.bError THEN
	stSystemStatus.nSystemStatus :=
		TO_INT(E_PlcSystemStatus.Error);
ELSIF bHoming THEN
	stSystemStatus.nSystemStatus :=
		TO_INT(E_PlcSystemStatus.Homing);
ELSIF nMovementStatus =
	TO_INT(E_PlcSystemStatus.Stopping) OR
	(bProtectiveStop AND NOT bControllerHalt) THEN
	stSystemStatus.nSystemStatus :=
		TO_INT(E_PlcSystemStatus.Stopping);
ELSIF stSystemStatus.bTarWorking THEN
	stSystemStatus.nSystemStatus :=
		TO_INT(E_PlcSystemStatus.Taring);
ELSE
	stSystemStatus.nSystemStatus := nMovementStatus;
END_IF

IF bSafetyError THEN
	stSystemStatus.nErrorCode := nSafetyErrorCode;
	stSystemStatus.nAxisErrorID := nSafetyAxisErrorID;
ELSIF bStartError THEN
	stSystemStatus.nErrorCode := nStartErrorCode;
	stSystemStatus.nAxisErrorID := 0;
ELSE
	stSystemStatus.nErrorCode := nMovementErrorCode;
	stSystemStatus.nAxisErrorID := nMovementAxisErrorID;
END_IF

END_FUNCTION_BLOCK

// ---- POUs/fb_BiaxialCoordinator.TcPOU
FUNCTION_BLOCK fb_BiaxialCoordinator
VAR_INPUT
	bStartRequest       : BOOL;
	bResetRequest       : BOOL;
	bAxesReady          : BOOL;
	bCommonAbortRequest : BOOL;
	bBusyX              : BOOL;
	bBusyY              : BOOL;
	bSavedPositionValidX: BOOL;
	bSavedPositionValidY: BOOL;
	nSyncPointX         : BYTE;
	nSyncPointY         : BYTE;
	nSyncCycleX         : INT;
	nSyncCycleY         : INT;
	bPeerAbortRequestX  : BOOL;
	bPeerAbortRequestY  : BOOL;
END_VAR

VAR_IN_OUT
	stCommandX : ST_MoveCommand;
	stCommandY : ST_MoveCommand;
END_VAR

VAR_OUTPUT
	bStartBoth      : BOOL;
	bSyncActive     : BOOL;
	bSyncRelease    : BOOL;
	bSingleCompleteX: BOOL;
	bSingleCompleteY: BOOL;
	bAbortX         : BOOL;
	bAbortY         : BOOL;
	bStartError     : BOOL;
	nStartErrorCode : UDINT;
END_VAR

VAR
	eState      : E_BiaxialState := E_BiaxialState.Idle;
END_VAR

VAR_TEMP
	bStartValid : BOOL;
END_VAR

VAR CONSTANT
	ERROR_BIAXIAL_START : UDINT := 2010;
END_VAR


// Pulse outputs are reset every scan. Abort outputs are deliberately retained
// while eState is Aborting.
bStartBoth := FALSE;
bSyncRelease := FALSE;
bSingleCompleteX := FALSE;
bSingleCompleteY := FALSE;

IF bResetRequest AND eState = E_BiaxialState.Idle THEN
	bStartError := FALSE;
	nStartErrorCode := 0;
END_IF

CASE eState OF
	E_BiaxialState.Idle:
		bSyncActive := FALSE;
		bAbortX := FALSE;
		bAbortY := FALSE;

		IF bStartRequest THEN
			// Preserve the established structural/compatibility checks. MATLAB
			// remains responsible for experiment-value validation.
			bStartValid :=
				bAxesReady AND
				stCommandX.nMode = 3 AND stCommandY.nMode = 3 AND
				stCommandX.nCycleCount >= 0 AND
				stCommandX.nCycleCount <= 50 AND
				stCommandY.nCycleCount >= 0 AND
				stCommandY.nCycleCount <= 50 AND
				stCommandX.nPreCycleCount >= 0 AND
				stCommandX.nPreCycleCount <= 50 AND
				stCommandY.nPreCycleCount >= 0 AND
				stCommandY.nPreCycleCount <= 50 AND
				stCommandX.nCycleCount = stCommandY.nCycleCount AND
				stCommandX.bIncludePreTest =
					stCommandY.bIncludePreTest AND
				stCommandX.bPreTestOnly = stCommandY.bPreTestOnly AND
				stCommandX.nPreCycleCount =
					stCommandY.nPreCycleCount AND
				stCommandX.bPreloadEnabled =
					stCommandY.bPreloadEnabled AND
				stCommandX.bPreUnloadToStart =
					stCommandY.bPreUnloadToStart AND
				stCommandX.nPostTestMode =
					stCommandY.nPostTestMode AND
				NOT (stCommandX.bPreTestOnly AND
					NOT stCommandX.bIncludePreTest);

			IF bStartValid THEN
				IF stCommandX.nPostTestMode < 0 OR
					stCommandX.nPostTestMode > 4 THEN
					bStartValid := FALSE;
				ELSIF stCommandX.nPostTestMode = 1 AND
					(NOT bSavedPositionValidX OR
					 NOT bSavedPositionValidY) THEN
					bStartValid := FALSE;
				ELSIF NOT stCommandX.bPreTestOnly AND
					stCommandX.nCycleCount = 0 AND
					((stCommandX.nStop1Mode < 1) OR
					 (stCommandX.nStop1Mode > 2) OR
					 (stCommandY.nStop1Mode < 1) OR
					 (stCommandY.nStop1Mode > 2) OR
					 (stCommandX.nStop2Mode < 0) OR
					 (stCommandX.nStop2Mode > 3) OR
					 (stCommandY.nStop2Mode < 0) OR
					 (stCommandY.nStop2Mode > 3)) THEN
					bStartValid := FALSE;
				ELSIF NOT stCommandX.bPreTestOnly AND
					stCommandX.nCycleCount > 0 AND
					((stCommandX.nLoadMode < 1) OR
					 (stCommandX.nLoadMode > 2) OR
					 (stCommandY.nLoadMode < 1) OR
					 (stCommandY.nLoadMode > 2) OR
					 (stCommandX.nUnloadMode < 1) OR
					 (stCommandX.nUnloadMode > 2) OR
					 (stCommandY.nUnloadMode < 1) OR
					 (stCommandY.nUnloadMode > 2)) THEN
					bStartValid := FALSE;
				END_IF
			END_IF

			IF bStartValid THEN
				bStartError := FALSE;
				nStartErrorCode := 0;
				bStartBoth := TRUE;
				bSyncActive := TRUE;
				eState := E_BiaxialState.Running;
			ELSE
				bStartError := TRUE;
				nStartErrorCode := ERROR_BIAXIAL_START;
			END_IF
		END_IF

	E_BiaxialState.Running:
		bSyncActive := TRUE;
		IF stCommandX.nCycleCount = 0 AND stCommandY.nCycleCount = 0 AND
			NOT stCommandX.bPreTestOnly THEN
			bSingleCompleteX :=
				nSyncPointY = TO_BYTE(E_SyncPoint.MainDone) AND
				nSyncPointX <> TO_BYTE(E_SyncPoint.MainDone);
			bSingleCompleteY :=
				nSyncPointX = TO_BYTE(E_SyncPoint.MainDone) AND
				nSyncPointY <> TO_BYTE(E_SyncPoint.MainDone);
		END_IF

		IF bCommonAbortRequest THEN
			bAbortX := TRUE;
			bAbortY := TRUE;
			eState := E_BiaxialState.Aborting;
		ELSIF bPeerAbortRequestX OR bPeerAbortRequestY THEN
			// A local relief request stops only the synchronized peer.
			bAbortX := bPeerAbortRequestY;
			bAbortY := bPeerAbortRequestX;
			eState := E_BiaxialState.Aborting;
		ELSIF nSyncPointX <> TO_BYTE(E_SyncPoint.None) AND
			nSyncPointX = nSyncPointY AND
			nSyncCycleX = nSyncCycleY THEN
			bSyncRelease := TRUE;
			IF nSyncPointX =
				TO_BYTE(E_SyncPoint.PostTestDone) THEN
				eState := E_BiaxialState.Completing;
			END_IF
		END_IF

	E_BiaxialState.Aborting:
		bSyncActive := TRUE;
		IF NOT bBusyX AND NOT bBusyY THEN
			bAbortX := FALSE;
			bAbortY := FALSE;
			bSyncActive := FALSE;
			eState := E_BiaxialState.Idle;
		END_IF

	E_BiaxialState.Completing:
		bSyncActive := TRUE;
		IF NOT bBusyX AND NOT bBusyY THEN
			bSyncActive := FALSE;
			eState := E_BiaxialState.Idle;
		END_IF
END_CASE

END_FUNCTION_BLOCK

// ---- POUs/fb_safety.TcPOU
FUNCTION_BLOCK fb_safety
VAR_INPUT
	bPower        : BOOL;
	bReset        : BOOL;
	bHalt         : BOOL;
	bHome         : BOOL;
	bRestoreReference : BOOL; // Static startup reference restore; no motion
	fRestoreReferencePosition : LREAL;
	bEndStopL     : BOOL; // TRUE when the normalized lower switch is active
	bEndStopH     : BOOL; // TRUE when the normalized upper switch is active
	bExternalBusy : BOOL; // Test motion or tare is active
END_VAR

VAR_OUTPUT
	bPowerStatus       : BOOL;
	bHaltDone          : BOOL;
	bError             : BOOL;
	nErrorCode         : UDINT;
	nAxisErrorID       : UDINT;
	bHoming            : BOOL;
	bHomed             : BOOL;
	bReferenceRestoreDone : BOOL;
	bReferenceRestoreBusy : BOOL;
	bStopped           : BOOL;
	bProtectiveStop    : BOOL; // Abort active test motion but retain commanded power
END_VAR

VAR_IN_OUT
	stAxis : AXIS_REF;
END_VAR

VAR
	fbPower        : MC_Power;
	fbReset        : MC_Reset;
	fbHalt         : MC_Halt;
	fbHome         : MC_Home;
	fbMoveToZero   : MC_MoveAbsolute;

	rtReset        : R_TRIG;
	rtHalt         : R_TRIG;
	rtHome         : R_TRIG;

	fbHomeTimeout  : TON;
	fbReferenceRestoreTimeout : TON;
	fbMoveTimeout  : TON;

	eState             : E_SafetyState := E_SafetyState.Idle;
	bFaultPowerInhibit : BOOL;
	bResetPending      : BOOL;
	bResetExecute      : BOOL;
	bHaltDonePulse     : BOOL;
	stHomeOptions      : ST_HomingOptions;
	fHomePosition      : LREAL;
	eHomingMode        : MC_HomingMode;
END_VAR

VAR CONSTANT
	HOME_PARK_POSITION : LREAL := 0.0;
	HOME_PARK_VELOCITY : LREAL := 5.0;
	HOME_TIMEOUT       : TIME := T#10M;
	REFERENCE_RESTORE_TIMEOUT : TIME := T#5S;
	REFERENCE_RESTORE_TOLERANCE : LREAL := 0.001;
	HOME_PARK_TIMEOUT  : TIME := T#10S;
	ERROR_POWER_FB       : UDINT := 1001;
	ERROR_RESET_FB       : UDINT := 1002;
	ERROR_HALT_FB        : UDINT := 1003;
	ERROR_HOME_FB        : UDINT := 1004;
	ERROR_AXIS           : UDINT := 1005;
	ERROR_LIMITS_CONFLICT: UDINT := 1006;
	ERROR_PARK_FB        : UDINT := 1008;
	ERROR_HOME_TIMEOUT   : UDINT := 1011;
	ERROR_PARK_TIMEOUT   : UDINT := 1012;
	ERROR_UPPER_LIMIT    : UDINT := 1013;
	ERROR_HOME_LIMIT     : UDINT := 1014;
	ERROR_HOME_COORDINATE: UDINT := 1015;
	ERROR_REFERENCE_RESTORE_TIMEOUT : UDINT := 1016;
	ERROR_REFERENCE_RESTORE_INVALID : UDINT := 1017;
END_VAR


// Commands are edge-triggered
rtReset(CLK := bReset);
rtHalt(CLK := bHalt);
rtHome(CLK := bHome);

// Halt completion is exposed as a one-cycle pulse.
bHaltDonePulse := FALSE;

// Retain reset until any active stop has returned the safety state to Idle.
IF rtReset.Q THEN
	bResetPending := TRUE;
END_IF
IF bResetPending AND eState = E_SafetyState.Idle THEN
	bResetPending := FALSE;
	IF bError THEN
		bResetExecute := TRUE;
	END_IF
END_IF

IF bResetExecute AND fbReset.Done THEN
	bResetExecute := FALSE;
	bError := FALSE;
	nErrorCode := 0;
	nAxisErrorID := 0;
	bFaultPowerInhibit := FALSE;
ELSIF bResetExecute AND fbReset.Error THEN
	bResetExecute := FALSE;
	bError := TRUE;
	nErrorCode := ERROR_RESET_FB;
	nAxisErrorID := fbReset.ErrorID;
	bFaultPowerInhibit := TRUE;
END_IF

// Latch genuine NC, wiring and motion-function-block faults
IF NOT bError THEN
	IF stAxis.Status.Error THEN
		bError := TRUE;
		nErrorCode := ERROR_AXIS;
		nAxisErrorID := stAxis.Status.ErrorID;
		eState := E_SafetyState.ErrorStop;
	ELSIF bEndStopL AND bEndStopH THEN
		bError := TRUE;
		nErrorCode := ERROR_LIMITS_CONFLICT;
		nAxisErrorID := 0;
		eState := E_SafetyState.ErrorStop;
	ELSIF fbPower.Error THEN
		bError := TRUE;
		nErrorCode := ERROR_POWER_FB;
		nAxisErrorID := fbPower.ErrorID;
		eState := E_SafetyState.ErrorStop;
	ELSIF fbHalt.Error THEN
		bError := TRUE;
		nErrorCode := ERROR_HALT_FB;
		nAxisErrorID := fbHalt.ErrorID;
		eState := E_SafetyState.ErrorStop;
	ELSIF fbHome.Error THEN
		bError := TRUE;
		nErrorCode := ERROR_HOME_FB;
		nAxisErrorID := fbHome.ErrorID;
		eState := E_SafetyState.ErrorStop;
	ELSIF fbMoveToZero.Error THEN
		bError := TRUE;
		nErrorCode := ERROR_PARK_FB;
		nAxisErrorID := fbMoveToZero.ErrorID;
		eState := E_SafetyState.ErrorStop;
	END_IF
END_IF

// Halt and switch to error stop
IF rtHalt.Q AND eState <> E_SafetyState.ErrorStop THEN
	eState := E_SafetyState.ProtectiveStop;
END_IF

CASE eState OF
	E_SafetyState.Idle:
		// Stop only when travelling farther into an active physical switch.
		IF (bEndStopL AND stAxis.Status.NegativeDirection) OR
			(bEndStopH AND stAxis.Status.PositiveDirection) THEN
			eState := E_SafetyState.ProtectiveStop;
		ELSIF rtHome.Q AND NOT bExternalBusy AND fbPower.Status THEN
			bReferenceRestoreDone := FALSE;
			eState := E_SafetyState.Homing;
		ELSIF bRestoreReference AND NOT bExternalBusy AND fbPower.Status THEN
			IF NOT ((fRestoreReferencePosition =
				fRestoreReferencePosition) AND
				ABS(fRestoreReferencePosition) < 1.0E300) THEN
				bError := TRUE;
				nErrorCode := ERROR_REFERENCE_RESTORE_INVALID;
				nAxisErrorID := 0;
				eState := E_SafetyState.ErrorStop;
			ELSE
				eState := E_SafetyState.RestoreReference;
			END_IF
		END_IF

	E_SafetyState.RestoreReference:
		IF fbReferenceRestoreTimeout.Q THEN
			bError := TRUE;
			nErrorCode := ERROR_REFERENCE_RESTORE_TIMEOUT;
			nAxisErrorID := 0;
			eState := E_SafetyState.ErrorStop;
		ELSIF fbHome.Done THEN
			eState := E_SafetyState.VerifyReference;
		END_IF

	E_SafetyState.VerifyReference:
		// ReadStatus() runs before this FB, so the scan after MC_Home.Done
		// verifies the NC result rather than trusting the retained value.
		IF fbReferenceRestoreTimeout.Q THEN
			bError := TRUE;
			nErrorCode := ERROR_REFERENCE_RESTORE_TIMEOUT;
			nAxisErrorID := 0;
			eState := E_SafetyState.ErrorStop;
		ELSIF NOT stAxis.Status.Homed OR
			ABS(stAxis.NcToPlc.ActPos -
				fRestoreReferencePosition) >
				REFERENCE_RESTORE_TOLERANCE THEN
			bError := TRUE;
			nErrorCode := ERROR_REFERENCE_RESTORE_INVALID;
			nAxisErrorID := 0;
			eState := E_SafetyState.ErrorStop;
		ELSE
			bReferenceRestoreDone := TRUE;
			eState := E_SafetyState.Complete;
		END_IF

	E_SafetyState.Homing:
		IF fbHomeTimeout.Q THEN
			bError := TRUE;
			nErrorCode := ERROR_HOME_TIMEOUT;
			nAxisErrorID := 0;
			eState := E_SafetyState.ErrorStop;
		ELSIF fbHome.Done THEN
			IF bEndStopL THEN
				bError := TRUE;
				nErrorCode := ERROR_HOME_LIMIT;
				nAxisErrorID := 0;
				eState := E_SafetyState.ErrorStop;
			ELSIF NOT stAxis.Status.Homed OR
				stAxis.NcToPlc.ActPos < -10.0 OR
				stAxis.NcToPlc.ActPos > 0.5 THEN
				// Reject an invalid coordinate instead of commanding a long move.
				bError := TRUE;
				nErrorCode := ERROR_HOME_COORDINATE;
				nAxisErrorID := 0;
				eState := E_SafetyState.ErrorStop;
			ELSE
				eState := E_SafetyState.MoveToZero;
			END_IF
		END_IF

	E_SafetyState.MoveToZero:
		IF stAxis.Status.NegativeDirection THEN
			// Parking from the lower reference toward zero must be positive.
			bError := TRUE;
			nErrorCode := ERROR_HOME_COORDINATE;
			nAxisErrorID := 0;
			eState := E_SafetyState.ErrorStop;
		ELSIF bEndStopH THEN
			bError := TRUE;
			nErrorCode := ERROR_UPPER_LIMIT;
			nAxisErrorID := 0;
			eState := E_SafetyState.ErrorStop;
		ELSIF fbMoveTimeout.Q THEN
			bError := TRUE;
			nErrorCode := ERROR_PARK_TIMEOUT;
			nAxisErrorID := 0;
			eState := E_SafetyState.ErrorStop;
		ELSIF fbMoveToZero.Done THEN
			eState := E_SafetyState.Complete;
		END_IF

	E_SafetyState.Complete:
		eState := E_SafetyState.Idle;

	E_SafetyState.ProtectiveStop:
		IF fbHalt.Done OR stAxis.Status.StandStill THEN
			bHaltDonePulse := TRUE;
			eState := E_SafetyState.Idle;
		END_IF

	E_SafetyState.ErrorStop:
		IF fbHalt.Done OR stAxis.Status.StandStill THEN
			bHaltDonePulse := TRUE;
			bFaultPowerInhibit := TRUE;
			eState := E_SafetyState.Idle;
		END_IF
END_CASE

fbHomeTimeout(
	IN := eState = E_SafetyState.Homing,
	PT := HOME_TIMEOUT);
fbReferenceRestoreTimeout(
	IN := eState = E_SafetyState.RestoreReference OR
		eState = E_SafetyState.VerifyReference,
	PT := REFERENCE_RESTORE_TIMEOUT);
fbMoveTimeout(
	IN := eState = E_SafetyState.MoveToZero,
	PT := HOME_PARK_TIMEOUT);

// Physical switches continuously block motion farther into the active limit
fbPower(
	Axis := stAxis,
	Enable := bPower AND NOT bFaultPowerInhibit,
	Enable_Positive := bPower AND NOT bFaultPowerInhibit AND NOT bEndStopH,
	Enable_Negative := bPower AND NOT bFaultPowerInhibit AND (NOT bEndStopL OR eState = E_SafetyState.Homing),
	Override := 100.0);

fbReset(
	Axis := stAxis,
	Execute := bResetExecute);

// Make both homing directions explicit:
// search toward the lower switch, then move positively away from it.
stHomeOptions.SearchDirection :=
	MC_Direction.MC_Negative_Direction;
stHomeOptions.SearchVelocity := 5;
stHomeOptions.SyncDirection :=
	MC_Direction.MC_Positive_Direction;
stHomeOptions.SyncVelocity := 2;
stHomeOptions.ReferenceMode :=
	E_EncoderReferenceMode.ENCODERREFERENCEMODE_PLCCAM;

// A retained startup coordinate uses MC_Direct, which changes the NC
// coordinate and referenced state without moving the motor. Normal homing
// continues to use the complete reference-cam search and release sequence.
IF eState = E_SafetyState.RestoreReference THEN
	fHomePosition := fRestoreReferencePosition;
	eHomingMode := MC_Direct;
	stHomeOptions.ClearPositionLag := TRUE;
ELSE
	fHomePosition := -5.0;
	eHomingMode := MC_DefaultHoming;
	stHomeOptions.ClearPositionLag := FALSE;
END_IF

fbHome(
	Axis := stAxis,
	Execute := eState = E_SafetyState.Homing OR
		eState = E_SafetyState.RestoreReference,
	Position := fHomePosition,
	HomingMode := eHomingMode,
	BufferMode := MC_Aborting,
	Options := stHomeOptions,
	bCalibrationCam := bEndStopL);

// Park at the safe working origin after TwinCAT has established the reference.
fbMoveToZero(
	Axis := stAxis,
	Execute := eState = E_SafetyState.MoveToZero,
	Position := HOME_PARK_POSITION,
	Velocity := HOME_PARK_VELOCITY,
	BufferMode := MC_Aborting);

fbHalt(
	Axis := stAxis,
	Execute := eState = E_SafetyState.ProtectiveStop OR
		eState = E_SafetyState.ErrorStop);

// Public status.
bPowerStatus := fbPower.Status;
bHaltDone := bHaltDonePulse OR fbHalt.Done;
bReferenceRestoreBusy :=
	eState = E_SafetyState.RestoreReference OR
	eState = E_SafetyState.VerifyReference;
bHoming := bReferenceRestoreBusy OR
	eState = E_SafetyState.Homing OR
	eState = E_SafetyState.MoveToZero;
bHomed := stAxis.Status.Homed;
bStopped := stAxis.Status.StandStill;
bProtectiveStop := eState = E_SafetyState.ProtectiveStop;

END_FUNCTION_BLOCK

// ---- POUs/fb_StatusBuffer.TcPOU
FUNCTION_BLOCK fb_StatusBuffer
VAR_IN_OUT
    stSystemStatus    : ST_SystemStatus;
    bStartTar         : BOOL;  // Cleared after completion or when tare is blocked
END_VAR
VAR_INPUT
	bBlockTar     : BOOL;  // Motion or homing is active

	// Tenzo buffer
    nRawTenzo    : DINT;
    fTenzoCons   : LREAL;
    fTenzoOffset : LREAL;
	
	// Position buffer
	fActPosition   : LREAL;
END_VAR
VAR
    fbStartTarRiseClp : R_TRIG;   // Detects the moment tare button is pressed
    bTarActive        : BOOL;     // Flag indicating taring is in progress
    nTarCounter       : INT;      // Counts up to 100 samples
    fTarAccumulator   : LREAL;    // Holds the running sum of samples
END_VAR
VAR_TEMP
    fCurrentCalculated: LREAL;    // Current force before the tare offset
	nNextHead        : INT;
END_VAR


// Calculate the current weight snapshot
fCurrentCalculated := (DINT_TO_LREAL(nRawTenzo) * fTenzoCons) + fTenzoOffset;

// Tare logic
// Reject a tare command received while motion or homing is active.
IF bStartTar AND bBlockTar THEN
	bStartTar := FALSE;
END_IF

fbStartTarRiseClp(CLK := bStartTar);

// Start the taring process
IF fbStartTarRiseClp.Q AND NOT bTarActive THEN
    bTarActive      := TRUE;
    nTarCounter     := 0;
    fTarAccumulator := 0.0;
END_IF

IF bTarActive THEN
    // Accumulate the current weight across 100 consecutive cycles
    fTarAccumulator := fTarAccumulator + fCurrentCalculated;
    nTarCounter     := nTarCounter + 1;
    
    // After 100 samples
    IF nTarCounter >= 100 THEN
        // Calculate the mean
        stSystemStatus.fTenzoTarOffset := - (fTarAccumulator / 100.0); 
        
        // Reset control flags
        bTarActive := FALSE;
        bStartTar  := FALSE;
    END_IF
END_IF

// Block movement while tare calculation is active.
stSystemStatus.bTarWorking := bTarActive;

// New head
nNextHead := stSystemStatus.nBufferHead + 1;
IF nNextHead > 50 THEN
    nNextHead := 1;
END_IF

// Buffering data
stSystemStatus.fTenzoBuffer[nNextHead] := fCurrentCalculated + stSystemStatus.fTenzoTarOffset;
stSystemStatus.fPosBuffer[nNextHead] := 50.0 - fActPosition;

// MATLAB status helpers
stSystemStatus.nBufferHead := nNextHead;
stSystemStatus.nSampleCounter := stSystemStatus.nSampleCounter + 1;

END_FUNCTION_BLOCK

// ---- POUs/MAIN.TcPOU
PROGRAM MAIN

VAR
	fbSafetyX : fb_safety;
	fbSafetyY : fb_safety;
	fbSystemBufferX : fb_StatusBuffer;
	fbSystemBufferY : fb_StatusBuffer;
	fbMovementControllerX : fb_MovementController;
	fbMovementControllerY : fb_MovementController;
	fbBiaxialCoordinator : fb_BiaxialCoordinator;
	fbStatusPublisherX : fb_AxisStatusPublisher;
	fbStatusPublisherY : fb_AxisStatusPublisher;
	
	// DUTs import
	stMoveCommandX : ST_MoveCommand;
	stMoveCommandY : ST_MoveCommand;

	stSystemStatusX : ST_SystemStatus;
	stSystemStatusY : ST_SystemStatus;

	stSettingsX : ST_Settings;
	stSettingsY : ST_Settings;

	// IO Links
    nRawTenzoX AT %I* : DINT;
	nRawTenzoY AT %I* : DINT;

	nEndStopLx AT %I* : BOOL;
	nEndStopHx AT %I* : BOOL;

	nEndStopLy AT %I* : BOOL;
	nEndStopHy AT %I* : BOOL;

	// Normalized physical limits: TRUE means that the switch is pressed.
	bEndStopLxActive : BOOL;
	bEndStopHxActive : BOOL;
	bEndStopLyActive : BOOL;
	bEndStopHyActive : BOOL;

	// PLC-owned synchronized start request
	bStartBiaxialTest : BOOL; // ADS one-shot after both axis commands are prepared

	// Persistent-axis checkpoint diagnostics. A successful checkpoint creates
	// an up-to-date Port_851.bootdata file before controller power is removed.
	bPersistentPositionSaved : BOOL;
	bPersistentPositionSaveBusy : BOOL;
	bPersistentPositionSaveError : BOOL;
	nPersistentPositionSaveErrorID : UDINT;
	nPersistentPositionCheckpointCounter : UDINT;

	fbWritePersistentData : FB_WritePersistentData;
	fbPersistentPositionSettle : TON;
	ftPowerRequestX : F_TRIG;
	ftPowerRequestY : F_TRIG;
	rtPersistentValidX : R_TRIG;
	rtPersistentValidY : R_TRIG;
	bPersistentInitialCheckpoint : BOOL := TRUE;
	bPersistentCheckpointPending : BOOL;
	bPersistentCheckpointInFlight : BOOL;
	bPersistentCheckpointStart : BOOL;
	bPersistentSafeToWrite : BOOL;
	nPersistentCheckpointRequestGeneration : UDINT;
	nPersistentCheckpointStartedGeneration : UDINT;
	nPersistentCheckpointCompletedGeneration : UDINT;
	fCheckpointPositionX : LREAL;
	fCheckpointPositionY : LREAL;
	bCheckpointValidX : BOOL;
	bCheckpointValidY : BOOL;

END_VAR

VAR_TEMP
	bBiaxialAxesReady : BOOL;
	bBiaxialCommonAbortRequest : BOOL;
	bRestoreReferenceX : BOOL;
	bRestoreReferenceY : BOOL;
END_VAR

////////////////////////////////
//////////   safety   //////////
////////////////////////////////

// Refresh NC status before making any safety or motion decision
GVL_Axis.xAxis.ReadStatus();
GVL_Axis.yAxis.ReadStatus();

// Requesting a physical home deliberately invalidates the old retained
// coordinate. Only a successfully referenced axis will make it valid again.
IF stMoveCommandX.bHome THEN
	GVL_Persistent.bLastPositionValidX := FALSE;
END_IF
IF stMoveCommandY.bHome THEN
	GVL_Persistent.bLastPositionValidY := FALSE;
END_IF

// On the first powered scan after a PLC/NC restart, statically restore each
// incremental axis to its last persistent coordinate. MC_Direct performs no
// motor movement. A normal reference-cam home always takes priority.
bRestoreReferenceX :=
	GVL_Persistent.bLastPositionValidX AND
	NOT GVL_Axis.xAxis.Status.Homed AND
	NOT fbSafetyX.bReferenceRestoreDone;
bRestoreReferenceY :=
	GVL_Persistent.bLastPositionValidY AND
	NOT GVL_Axis.yAxis.Status.Homed AND
	NOT fbSafetyY.bReferenceRestoreDone;

// Normalize the active-low physical switches
bEndStopLxActive := NOT nEndStopLx;
bEndStopHxActive := NOT nEndStopHx;
bEndStopLyActive := NOT nEndStopLy;
bEndStopHyActive := NOT nEndStopHy;

fbSafetyX(
    stAxis := GVL_Axis.xAxis,
    bPower := stMoveCommandX.bPower,
    bReset := stMoveCommandX.bReset,
    bHalt := stMoveCommandX.bHalt OR fbMovementControllerX.stateHalt,
    bHome := stMoveCommandX.bHome,
	bRestoreReference := bRestoreReferenceX,
	fRestoreReferencePosition := GVL_Persistent.fLastPositionX,
    bEndStopL := bEndStopLxActive,
	bEndStopH := bEndStopHxActive,
	bExternalBusy := fbMovementControllerX.bBusy OR stSystemStatusX.bTarWorking
);

fbSafetyY(
    stAxis := GVL_Axis.yAxis,
    bPower := stMoveCommandY.bPower,
    bReset := stMoveCommandY.bReset,
    bHalt := stMoveCommandY.bHalt OR fbMovementControllerY.stateHalt,
    bHome := stMoveCommandY.bHome,
	bRestoreReference := bRestoreReferenceY,
	fRestoreReferencePosition := GVL_Persistent.fLastPositionY,
    bEndStopL := bEndStopLyActive,
	bEndStopH := bEndStopHyActive,
	bExternalBusy := fbMovementControllerY.bBusy OR stSystemStatusY.bTarWorking
);

////////////////////////////////
////////// Update data /////////
////////////////////////////////

fbSystemBufferX(
	stSystemStatus:= stSystemStatusX,
	bBlockTar:= fbMovementControllerX.bBusy OR fbSafetyX.bHoming OR
		NOT fbSafetyX.bHomed,
	nRawTenzo:= -nRawTenzoX,
	fTenzoCons:=stSettingsX.fTenzoCons,
	fTenzoOffset:= stSettingsX.fTenzoOffset,
	bStartTar:= stMoveCommandX.bStartTar,
	fActPosition:= GVL_Axis.xAxis.NcToPlc.ActPos);
	
fbSystemBufferY(
	stSystemStatus:= stSystemStatusY,
	bBlockTar:= fbMovementControllerY.bBusy OR fbSafetyY.bHoming OR
		NOT fbSafetyY.bHomed,
	nRawTenzo:= nRawTenzoY,
	fTenzoCons:=stSettingsY.fTenzoCons,
	fTenzoOffset:= stSettingsY.fTenzoOffset,
	bStartTar:= stMoveCommandY.bStartTar,
	fActPosition:= GVL_Axis.yAxis.NcToPlc.ActPos);

/////////////////////////////////////
////////// Main Move Logic //////////
/////////////////////////////////////

// A shared request starts both axes in one PLC scan. Single-axis tests keep
// using their individual bExecute fields and never enable synchronization.
bBiaxialAxesReady :=
	NOT fbMovementControllerX.bBusy AND
	NOT fbMovementControllerY.bBusy AND
	NOT fbMovementControllerX.bError AND
	NOT fbMovementControllerY.bError AND
	NOT fbSafetyX.bError AND NOT fbSafetyY.bError AND
	NOT fbSafetyX.bHoming AND NOT fbSafetyY.bHoming AND
	fbSafetyX.bHomed AND fbSafetyY.bHomed AND
	NOT stSystemStatusX.bTarWorking AND
	NOT stSystemStatusY.bTarWorking AND
	fbSafetyX.bPowerStatus AND fbSafetyY.bPowerStatus;

// Ignore ProtectiveStop when it was produced by the controller's own
// controlled halt. Operator, end-stop and independent safety stops abort both
// axes; an overforce relief request aborts only the synchronized peer.
bBiaxialCommonAbortRequest :=
	fbMovementControllerX.bError OR fbMovementControllerY.bError OR
	fbSafetyX.bError OR fbSafetyY.bError OR
	(fbSafetyX.bProtectiveStop AND
	 NOT fbMovementControllerX.stateHalt) OR
	(fbSafetyY.bProtectiveStop AND
	 NOT fbMovementControllerY.stateHalt) OR
	(bEndStopLxActive AND GVL_Axis.xAxis.Status.NegativeDirection) OR
	(bEndStopHxActive AND GVL_Axis.xAxis.Status.PositiveDirection) OR
	(bEndStopLyActive AND GVL_Axis.yAxis.Status.NegativeDirection) OR
	(bEndStopHyActive AND GVL_Axis.yAxis.Status.PositiveDirection) OR
	stMoveCommandX.bHalt OR stMoveCommandY.bHalt;

fbBiaxialCoordinator(
	bStartRequest := bStartBiaxialTest,
	bResetRequest := stMoveCommandX.bReset OR stMoveCommandY.bReset,
	bAxesReady := bBiaxialAxesReady,
	bCommonAbortRequest := bBiaxialCommonAbortRequest,
	bBusyX := fbMovementControllerX.bBusy,
	bBusyY := fbMovementControllerY.bBusy,
	bSavedPositionValidX := fbMovementControllerX.bSavedPositionValid,
	bSavedPositionValidY := fbMovementControllerY.bSavedPositionValid,
	nSyncPointX := fbMovementControllerX.nSyncPoint,
	nSyncPointY := fbMovementControllerY.nSyncPoint,
	nSyncCycleX := fbMovementControllerX.nSyncCycle,
	nSyncCycleY := fbMovementControllerY.nSyncCycle,
	bPeerAbortRequestX := fbMovementControllerX.bPeerAbortRequest,
	bPeerAbortRequestY := fbMovementControllerY.bPeerAbortRequest,
	stCommandX := stMoveCommandX,
	stCommandY := stMoveCommandY);

IF bStartBiaxialTest THEN
	bStartBiaxialTest := FALSE;
END_IF

IF fbBiaxialCoordinator.bStartBoth THEN
	stMoveCommandX.bExecute := TRUE;
	stMoveCommandY.bExecute := TRUE;
END_IF

fbMovementControllerX(
	Axis := GVL_Axis.xAxis,
	stMoveCommand := stMoveCommandX,
	stSettings := stSettingsX,
	fActPosition := GVL_Axis.xAxis.NcToPlc.ActPos,
    bPowerState := fbSafetyX.bPowerStatus,
	bHaltDone := fbSafetyX.bHaltDone,
	bAxisStopped := fbSafetyX.bStopped,
	bSafetyError := fbSafetyX.bError,
	bProtectiveStop := fbSafetyX.bProtectiveStop,
	bExternalBusy := fbSafetyX.bHoming OR
		NOT fbSafetyX.bHomed OR stSystemStatusX.bTarWorking,
	bReferenceValid := fbSafetyX.bHomed,
	bInvalidateSavedPosition := stMoveCommandX.bHome,
	bSyncEnabled := fbBiaxialCoordinator.bSyncActive,
	bSyncRelease := fbBiaxialCoordinator.bSyncRelease,
	bSyncAbort := fbBiaxialCoordinator.bAbortX,
	bSyncSingleComplete := fbBiaxialCoordinator.bSingleCompleteX,
    fForce := stSystemStatusX.fTenzoBuffer[stSystemStatusX.nBufferHead]);

fbMovementControllerY(
	Axis := GVL_Axis.yAxis,
	stMoveCommand := stMoveCommandY,
	stSettings := stSettingsY,
	fActPosition := GVL_Axis.yAxis.NcToPlc.ActPos,
    bPowerState := fbSafetyY.bPowerStatus,
	bHaltDone := fbSafetyY.bHaltDone,
	bAxisStopped := fbSafetyY.bStopped,
	bSafetyError := fbSafetyY.bError,
	bProtectiveStop := fbSafetyY.bProtectiveStop,
	bExternalBusy := fbSafetyY.bHoming OR
		NOT fbSafetyY.bHomed OR stSystemStatusY.bTarWorking,
	bReferenceValid := fbSafetyY.bHomed,
	bInvalidateSavedPosition := stMoveCommandY.bHome,
	bSyncEnabled := fbBiaxialCoordinator.bSyncActive,
	bSyncRelease := fbBiaxialCoordinator.bSyncRelease,
	bSyncAbort := fbBiaxialCoordinator.bAbortY,
	bSyncSingleComplete := fbBiaxialCoordinator.bSingleCompleteY,
	fForce := stSystemStatusY.fTenzoBuffer[stSystemStatusY.nBufferHead]);

///////////////////////////////////////////////////
////// ADS status contract for each axis //////////
///////////////////////////////////////////////////

fbStatusPublisherX(
	fActPosition := GVL_Axis.xAxis.NcToPlc.ActPos,
	bPowerStatus := fbSafetyX.bPowerStatus,
	bHoming := fbSafetyX.bHoming,
	bHomed := fbSafetyX.bHomed,
	bStopped := fbSafetyX.bStopped,
	bProtectiveStop := fbSafetyX.bProtectiveStop,
	bControllerHalt := fbMovementControllerX.stateHalt,
	bSafetyError := fbSafetyX.bError,
	nSafetyErrorCode := fbSafetyX.nErrorCode,
	nSafetyAxisErrorID := fbSafetyX.nAxisErrorID,
	bMovementBusy := fbMovementControllerX.bBusy,
	bMovementError := fbMovementControllerX.bError,
	nMovementStatus := fbMovementControllerX.nSystemStatus,
	nMovementErrorCode := fbMovementControllerX.nErrorCode,
	nMovementAxisErrorID := fbMovementControllerX.nAxisErrorID,
	nOperationCounter := fbMovementControllerX.nOperationCounter,
	bSavedPositionValid := fbMovementControllerX.bSavedPositionValid,
	bStartError := fbBiaxialCoordinator.bStartError,
	nStartErrorCode := fbBiaxialCoordinator.nStartErrorCode,
	stSystemStatus := stSystemStatusX);

fbStatusPublisherY(
	fActPosition := GVL_Axis.yAxis.NcToPlc.ActPos,
	bPowerStatus := fbSafetyY.bPowerStatus,
	bHoming := fbSafetyY.bHoming,
	bHomed := fbSafetyY.bHomed,
	bStopped := fbSafetyY.bStopped,
	bProtectiveStop := fbSafetyY.bProtectiveStop,
	bControllerHalt := fbMovementControllerY.stateHalt,
	bSafetyError := fbSafetyY.bError,
	nSafetyErrorCode := fbSafetyY.nErrorCode,
	nSafetyAxisErrorID := fbSafetyY.nAxisErrorID,
	bMovementBusy := fbMovementControllerY.bBusy,
	bMovementError := fbMovementControllerY.bError,
	nMovementStatus := fbMovementControllerY.nSystemStatus,
	nMovementErrorCode := fbMovementControllerY.nErrorCode,
	nMovementAxisErrorID := fbMovementControllerY.nAxisErrorID,
	nOperationCounter := fbMovementControllerY.nOperationCounter,
	bSavedPositionValid := fbMovementControllerY.bSavedPositionValid,
	bStartError := fbBiaxialCoordinator.bStartError,
	nStartErrorCode := fbBiaxialCoordinator.nStartErrorCode,
	stSystemStatus := stSystemStatusY);

// Track the last valid coordinate continuously in persistent PLC memory.
// Values are never replaced while an axis is unreferenced, homing, or in an
// NC error, so startup cannot accidentally retain the raw zero coordinate.
IF fbSafetyX.bHomed AND NOT fbSafetyX.bHoming AND
	NOT GVL_Axis.xAxis.Status.Error AND
	(GVL_Axis.xAxis.NcToPlc.ActPos =
		GVL_Axis.xAxis.NcToPlc.ActPos) AND
	ABS(GVL_Axis.xAxis.NcToPlc.ActPos) < 1.0E300 THEN
	GVL_Persistent.fLastPositionX :=
		GVL_Axis.xAxis.NcToPlc.ActPos;
	GVL_Persistent.bLastPositionValidX := TRUE;
END_IF

IF fbSafetyY.bHomed AND NOT fbSafetyY.bHoming AND
	NOT GVL_Axis.yAxis.Status.Error AND
	(GVL_Axis.yAxis.NcToPlc.ActPos =
		GVL_Axis.yAxis.NcToPlc.ActPos) AND
	ABS(GVL_Axis.yAxis.NcToPlc.ActPos) < 1.0E300 THEN
	GVL_Persistent.fLastPositionY :=
		GVL_Axis.yAxis.NcToPlc.ActPos;
	GVL_Persistent.bLastPositionValidY := TRUE;
END_IF

///////////////////////////////////////////////////
//// Persistent coordinate disk checkpoint ///////
///////////////////////////////////////////////////

// PERSISTENT values in RAM are normally copied to Port_851.bootdata only on
// an orderly TwinCAT stop. Create a checkpoint after a normal home and when
// the operator removes commanded motor power so a later hard power-off does
// not fall back to an older coordinate. Never write continuously while the
// axes move; that would both save an unsafe intermediate coordinate and wear
// the controller's flash storage.
ftPowerRequestX(CLK := stMoveCommandX.bPower);
ftPowerRequestY(CLK := stMoveCommandY.bPower);
rtPersistentValidX(CLK := GVL_Persistent.bLastPositionValidX);
rtPersistentValidY(CLK := GVL_Persistent.bLastPositionValidY);

IF bPersistentInitialCheckpoint OR ftPowerRequestX.Q OR
	ftPowerRequestY.Q OR rtPersistentValidX.Q OR
	rtPersistentValidY.Q THEN
	bPersistentCheckpointPending := TRUE;
	nPersistentCheckpointRequestGeneration :=
		nPersistentCheckpointRequestGeneration + 1;
	bPersistentPositionSaved := FALSE;
	bPersistentPositionSaveError := FALSE;
	nPersistentPositionSaveErrorID := 0;
	bPersistentInitialCheckpoint := FALSE;
END_IF

// Mark the public diagnostic false as soon as a referenced coordinate moves
// away from the last successfully written snapshot. A new disk write remains
// intentionally tied to home/power-off rather than every test endpoint.
IF bPersistentPositionSaved AND (
	(GVL_Persistent.bLastPositionValidX <>
		bCheckpointValidX) OR
	(GVL_Persistent.bLastPositionValidY <>
		bCheckpointValidY) OR
	(GVL_Persistent.bLastPositionValidX AND
		ABS(GVL_Persistent.fLastPositionX -
			fCheckpointPositionX) > 0.001) OR
	(GVL_Persistent.bLastPositionValidY AND
		ABS(GVL_Persistent.fLastPositionY -
			fCheckpointPositionY) > 0.001)) THEN
	bPersistentPositionSaved := FALSE;
END_IF

// Wait for a stable non-moving state before writing. An already loaded
// persistent coordinate may be checkpointed while its axis is unpowered; if
// powered, the NC axis must be referenced, stopped and error-free.
bPersistentSafeToWrite :=
	(GVL_Persistent.bLastPositionValidX OR
		GVL_Persistent.bLastPositionValidY) AND
	NOT fbMovementControllerX.bBusy AND
	NOT fbMovementControllerY.bBusy AND
	NOT fbSafetyX.bHoming AND NOT fbSafetyY.bHoming AND
	NOT stSystemStatusX.bTarWorking AND
	NOT stSystemStatusY.bTarWorking AND
	(NOT fbSafetyX.bPowerStatus OR
		(fbSafetyX.bHomed AND fbSafetyX.bStopped AND
			NOT GVL_Axis.xAxis.Status.Error)) AND
	(NOT fbSafetyY.bPowerStatus OR
		(fbSafetyY.bHomed AND fbSafetyY.bStopped AND
			NOT GVL_Axis.yAxis.Status.Error));

fbPersistentPositionSettle(
	IN := bPersistentCheckpointPending AND
		NOT bPersistentCheckpointInFlight AND
		bPersistentSafeToWrite,
	PT := T#1S);

bPersistentCheckpointStart :=
	fbPersistentPositionSettle.Q AND
	NOT fbWritePersistentData.BUSY AND
	NOT bPersistentCheckpointInFlight;

fbWritePersistentData(
	NETID := '',
	PORT := TwinCAT_SystemInfoVarList._AppInfo.AdsPort,
	START := bPersistentCheckpointStart,
	TMOUT := T#5S,
	MODE := SPDM_VAR_BOOST);

